// TwinCAT 3 PLC project M3V3_UltraCap
// ProgramVersion: 3.1.4023.0
// libraries:
//   Tc2_Standard, * (Beckhoff Automation GmbH)
//   Tc2_System, * (Beckhoff Automation GmbH)
//   Tc2_Utilities, * (Beckhoff Automation GmbH)
//   Tc3_EventLogger, * (Beckhoff Automation GmbH)
//   Tc3_Module, * (Beckhoff Automation GmbH)
// project tree:
//   DUTs/ E_ChargerType.TcDUT (not stored), E_State.TcDUT (not stored), E_VoltFB.TcDUT (not stored), ST_Alarm_Base.TcDUT (not stored), ST_canRxdata.TcDUT, ST_Cap_Base.TcDUT, ST_Charger_Base.TcDUT, ST_ChargeTime.TcDUT (not stored), ST_MagDriver.TcDUT, ST_Module.TcDUT, ST_PB_Base.TcDUT, ST_Segment_Base.TcDUT, ST_Setpoints_Base.TcDUT, ST_UCDevices.TcDUT, ST_UC_Status.TcDUT, ST_UC_Status_Dummy.TcDUT, ST_UC_Trip_Base.TcDUT, ST_VoltMon_Base.TcDUT (not stored), ST_VoltTran_Base.TcDUT
//   GVLs/ Alarms_DB.TcGVL, ChargeTime_DB.TcGVL, csv_DB.TcGVL (not stored), GVL.TcGVL, plc_plc_comm_DB.TcGVL, HMI_DB.TcGVL, Input.TcGVL, LV.TcGVL, MCP_IO.TcGVL, Output.TcGVL, Permissives_DB.TcGVL, Setpoints.TcGVL, Trips_DB.TcGVL (not stored)
//   / PlcTask.TcTTO (not stored)
//   POUs/ ADC_10V.TcPOU (not stored), ADC_5V.TcPOU (not stored), Alarms.TcPOU, Alarms_FB.TcPOU (not stored), Alias.TcPOU, AnalogConversion.TcPOU, AQ.TcPOU (not stored), CAN_comm.TcPOU, ChargeTime.TcPOU, Heartbeat.TcPOU, HMI.TcPOU, LCA_CAL.TcPOU, MAIN.TcPOU, Norm_x.TcPOU (not stored), Permissives.TcPOU, plc_plc_comm.TcPOU, RW_CSV.TcPOU, Stagger_FB.TcPOU (not stored), Sequence.TcPOU, VoltageMonitor.TcPOU, VoltMonAC_FB.TcPOU (not stored), VoltTranBd.TcPOU
//   POUs/csv/ P_ArgToConvExample.TcPOU, P_StringToConvExample.TcPOU, P_TextModeRead.TcPOU, P_TextModeWrite.TcPOU, P_TextModeWrite_og.TcPOU
// real-time tasks:
//   TASK PlcTask: cycle T#10ms, priority 20, ADS port 350
// I/O:
//   DEVICE Device 3 (EtherCAT), AmsNetId 5.107.220.56.4.1
//     Term 1 (EK1101) [EK1101 EtherCAT Coupler (2A E-Bus, ID switch)]
//       Term 2 (EL3068) [EL3068 8K. Ana. Eingang 0-10V]
//       Term 3 (EL3068) [EL3068 8K. Ana. Eingang 0-10V]
//       Term 4 (EL1008) [EL1008 8Ch. Dig. Input 24V, 3ms]
//       Term 5 (EL1008) [EL1008 8Ch. Dig. Input 24V, 3ms]
//       Term 6 (EL2008) [EL2008 8Ch. Dig. Output 24V, 0.5A]
//       Term 7 (EL2008) [EL2008 8Ch. Dig. Output 24V, 0.5A]
//       Term 8 (EL1008) [EL1008 8Ch. Dig. Input 24V, 3ms]
//       Term 9 (EL2008) [EL2008 8Ch. Dig. Output 24V, 0.5A]
//       Term 10 (EL4008) [EL4008 8Ch. Ana. Output 0-10V, 12bit]
//       Term 21 (EL6751) [EL6751 CANopen Master]
//       Term 22 (EL9011) [EL9011 End Terminal]
//   DEVICE Device 1 (EL6751), AmsNetId 5.107.220.56.2.1
//     Vector__XXX
// variable links:
//   M3V3_UltraCap/M3V3_UltraCap Instance <-> Device 1 (EL6751)/Prepared DBC Signals/Vector__XXX/ElectricalData01
//     PlcTask Inputs/Input.R1_10_CapNumber[1]/Elec_AveVolt <-> Message_Inputs/ELECTRICAL_AVERAGE_VOLTAGE
//     PlcTask Inputs/Input.R1_10_CapNumber[1]/Elec_Balancing <-> Message_Inputs/ELECTRICAL_STATUS_BALANCING
//     PlcTask Inputs/Input.R1_10_CapNumber[1]/Elec_HighestVolt <-> Message_Inputs/ELECTRICAL_HIGHEST_VOLTAGE
//     PlcTask Inputs/Input.R1_10_CapNumber[1]/Elec_Imbalance <-> Message_Inputs/ELECTRICAL_STATUS_IMBALANCE
//     PlcTask Inputs/Input.R1_10_CapNumber[1]/Elec_OverVoltage <-> Message_Inputs/ELECTRICAL_STATUS_OVERVOLTAGE
//     PlcTask Inputs/Input.R1_10_CapNumber[1]/Elec_VoltageSum <-> Message_Inputs/ELECTRICAL_VOLTAGE_SUM
//   M3V3_UltraCap/M3V3_UltraCap Instance <-> Device 1 (EL6751)/Prepared DBC Signals/Vector__XXX/ElectricalData02
//     PlcTask Inputs/Input.R1_10_CapNumber[2]/Elec_AveVolt <-> Message_Inputs/ELECTRICAL_AVERAGE_VOLTAGE
//     PlcTask Inputs/Input.R1_10_CapNumber[2]/Elec_Balancing <-> Message_Inputs/ELECTRICAL_STATUS_BALANCING
//     PlcTask Inputs/Input.R1_10_CapNumber[2]/Elec_HighestVolt <-> Message_Inputs/ELECTRICAL_HIGHEST_VOLTAGE
//     PlcTask Inputs/Input.R1_10_CapNumber[2]/Elec_Imbalance <-> Message_Inputs/ELECTRICAL_STATUS_IMBALANCE
//     PlcTask Inputs/Input.R1_10_CapNumber[2]/Elec_OverVoltage <-> Message_Inputs/ELECTRICAL_STATUS_OVERVOLTAGE
//     PlcTask Inputs/Input.R1_10_CapNumber[2]/Elec_VoltageSum <-> Message_Inputs/ELECTRICAL_VOLTAGE_SUM
//   M3V3_UltraCap/M3V3_UltraCap Instance <-> Device 1 (EL6751)/Prepared DBC Signals/Vector__XXX/ElectricalData03
//     PlcTask Inputs/Input.R1_10_CapNumber[3]/Elec_AveVolt <-> Message_Inputs/ELECTRICAL_AVERAGE_VOLTAGE
//     PlcTask Inputs/Input.R1_10_CapNumber[3]/Elec_Balancing <-> Message_Inputs/ELECTRICAL_STATUS_BALANCING
//     PlcTask Inputs/Input.R1_10_CapNumber[3]/Elec_HighestVolt <-> Message_Inputs/ELECTRICAL_HIGHEST_VOLTAGE
//     PlcTask Inputs/Input.R1_10_CapNumber[3]/Elec_Imbalance <-> Message_Inputs/ELECTRICAL_STATUS_IMBALANCE
//     PlcTask Inputs/Input.R1_10_CapNumber[3]/Elec_OverVoltage <-> Message_Inputs/ELECTRICAL_STATUS_OVERVOLTAGE
//     PlcTask Inputs/Input.R1_10_CapNumber[3]/Elec_VoltageSum <-> Message_Inputs/ELECTRICAL_VOLTAGE_SUM
//   M3V3_UltraCap/M3V3_UltraCap Instance <-> Device 1 (EL6751)/Prepared DBC Signals/Vector__XXX/ElectricalData04
//     PlcTask Inputs/Input.R1_10_CapNumber[4]/Elec_AveVolt <-> Message_Inputs/ELECTRICAL_AVERAGE_VOLTAGE
//     PlcTask Inputs/Input.R1_10_CapNumber[4]/Elec_Balancing <-> Message_Inputs/ELECTRICAL_STATUS_BALANCING
//     PlcTask Inputs/Input.R1_10_CapNumber[4]/Elec_HighestVolt <-> Message_Inputs/ELECTRICAL_HIGHEST_VOLTAGE
//     PlcTask Inputs/Input.R1_10_CapNumber[4]/Elec_Imbalance <-> Message_Inputs/ELECTRICAL_STATUS_IMBALANCE
//     PlcTask Inputs/Input.R1_10_CapNumber[4]/Elec_OverVoltage <-> Message_Inputs/ELECTRICAL_STATUS_OVERVOLTAGE
//     PlcTask Inputs/Input.R1_10_CapNumber[4]/Elec_VoltageSum <-> Message_Inputs/ELECTRICAL_VOLTAGE_SUM
//   M3V3_UltraCap/M3V3_UltraCap Instance <-> Device 1 (EL6751)/Prepared DBC Signals/Vector__XXX/ElectricalData05
//     PlcTask Inputs/Input.R1_10_CapNumber[5]/Elec_AveVolt <-> Message_Inputs/ELECTRICAL_AVERAGE_VOLTAGE
//     PlcTask Inputs/Input.R1_10_CapNumber[5]/Elec_Balancing <-> Message_Inputs/ELECTRICAL_STATUS_BALANCING
//     PlcTask Inputs/Input.R1_10_CapNumber[5]/Elec_HighestVolt <-> Message_Inputs/ELECTRICAL_HIGHEST_VOLTAGE
//     PlcTask Inputs/Input.R1_10_CapNumber[5]/Elec_Imbalance <-> Message_Inputs/ELECTRICAL_STATUS_IMBALANCE
//     PlcTask Inputs/Input.R1_10_CapNumber[5]/Elec_OverVoltage <-> Message_Inputs/ELECTRICAL_STATUS_OVERVOLTAGE
//     PlcTask Inputs/Input.R1_10_CapNumber[5]/Elec_VoltageSum <-> Message_Inputs/ELECTRICAL_VOLTAGE_SUM
//   M3V3_UltraCap/M3V3_UltraCap Instance <-> Device 1 (EL6751)/Prepared DBC Signals/Vector__XXX/ElectricalData06
//     PlcTask Inputs/Input.R1_10_CapNumber[6]/Elec_AveVolt <-> Message_Inputs/ELECTRICAL_AVERAGE_VOLTAGE
//     PlcTask Inputs/Input.R1_10_CapNumber[6]/Elec_Balancing <-> Message_Inputs/ELECTRICAL_STATUS_BALANCING
//     PlcTask Inputs/Input.R1_10_CapNumber[6]/Elec_HighestVolt <-> Message_Inputs/ELECTRICAL_HIGHEST_VOLTAGE
//     PlcTask Inputs/Input.R1_10_CapNumber[6]/Elec_Imbalance <-> Message_Inputs/ELECTRICAL_STATUS_IMBALANCE
//     PlcTask Inputs/Input.R1_10_CapNumber[6]/Elec_OverVoltage <-> Message_Inputs/ELECTRICAL_STATUS_OVERVOLTAGE
//     PlcTask Inputs/Input.R1_10_CapNumber[6]/Elec_VoltageSum <-> Message_Inputs/ELECTRICAL_VOLTAGE_SUM
//   M3V3_UltraCap/M3V3_UltraCap Instance <-> Device 1 (EL6751)/Prepared DBC Signals/Vector__XXX/ElectricalData07
//     PlcTask Inputs/Input.R1_10_CapNumber[7]/Elec_AveVolt <-> Message_Inputs/ELECTRICAL_AVERAGE_VOLTAGE
//     PlcTask Inputs/Input.R1_10_CapNumber[7]/Elec_Balancing <-> Message_Inputs/ELECTRICAL_STATUS_BALANCING
//     PlcTask Inputs/Input.R1_10_CapNumber[7]/Elec_HighestVolt <-> Message_Inputs/ELECTRICAL_HIGHEST_VOLTAGE
//     PlcTask Inputs/Input.R1_10_CapNumber[7]/Elec_Imbalance <-> Message_Inputs/ELECTRICAL_STATUS_IMBALANCE
//     PlcTask Inputs/Input.R1_10_CapNumber[7]/Elec_OverVoltage <-> Message_Inputs/ELECTRICAL_STATUS_OVERVOLTAGE
//     PlcTask Inputs/Input.R1_10_CapNumber[7]/Elec_VoltageSum <-> Message_Inputs/ELECTRICAL_VOLTAGE_SUM
//   M3V3_UltraCap/M3V3_UltraCap Instance <-> Device 1 (EL6751)/Prepared DBC Signals/Vector__XXX/ElectricalData08
//     PlcTask Inputs/Input.R1_10_CapNumber[8]/Elec_AveVolt <-> Message_Inputs/ELECTRICAL_AVERAGE_VOLTAGE
//     PlcTask Inputs/Input.R1_10_CapNumber[8]/Elec_Balancing <-> Message_Inputs/ELECTRICAL_STATUS_BALANCING
//     PlcTask Inputs/Input.R1_10_CapNumber[8]/Elec_HighestVolt <-> Message_Inputs/ELECTRICAL_HIGHEST_VOLTAGE
//     PlcTask Inputs/Input.R1_10_CapNumber[8]/Elec_Imbalance <-> Message_Inputs/ELECTRICAL_STATUS_IMBALANCE
//     PlcTask Inputs/Input.R1_10_CapNumber[8]/Elec_OverVoltage <-> Message_Inputs/ELECTRICAL_STATUS_OVERVOLTAGE
//     PlcTask Inputs/Input.R1_10_CapNumber[8]/Elec_VoltageSum <-> Message_Inputs/ELECTRICAL_VOLTAGE_SUM
//   M3V3_UltraCap/M3V3_UltraCap Instance <-> Device 1 (EL6751)/Prepared DBC Signals/Vector__XXX/ElectricalData09
//     PlcTask Inputs/Input.R1_10_CapNumber[9]/Elec_AveVolt <-> Message_Inputs/ELECTRICAL_AVERAGE_VOLTAGE
//     PlcTask Inputs/Input.R1_10_CapNumber[9]/Elec_Balancing <-> Message_Inputs/ELECTRICAL_STATUS_BALANCING
//     PlcTask Inputs/Input.R1_10_CapNumber[9]/Elec_HighestVolt <-> Message_Inputs/ELECTRICAL_HIGHEST_VOLTAGE
//     PlcTask Inputs/Input.R1_10_CapNumber[9]/Elec_Imbalance <-> Message_Inputs/ELECTRICAL_STATUS_IMBALANCE
//     PlcTask Inputs/Input.R1_10_CapNumber[9]/Elec_OverVoltage <-> Message_Inputs/ELECTRICAL_STATUS_OVERVOLTAGE
//     PlcTask Inputs/Input.R1_10_CapNumber[9]/Elec_VoltageSum <-> Message_Inputs/ELECTRICAL_VOLTAGE_SUM
//   M3V3_UltraCap/M3V3_UltraCap Instance <-> Device 1 (EL6751)/Prepared DBC Signals/Vector__XXX/ElectricalData0A
//     PlcTask Inputs/Input.R1_10_CapNumber[10]/Elec_AveVolt <-> Message_Inputs/ELECTRICAL_AVERAGE_VOLTAGE
//     PlcTask Inputs/Input.R1_10_CapNumber[10]/Elec_Balancing <-> Message_Inputs/ELECTRICAL_STATUS_BALANCING
//     PlcTask Inputs/Input.R1_10_CapNumber[10]/Elec_HighestVolt <-> Message_Inputs/ELECTRICAL_HIGHEST_VOLTAGE
//     PlcTask Inputs/Input.R1_10_CapNumber[10]/Elec_Imbalance <-> Message_Inputs/ELECTRICAL_STATUS_IMBALANCE
//     PlcTask Inputs/Input.R1_10_CapNumber[10]/Elec_OverVoltage <-> Message_Inputs/ELECTRICAL_STATUS_OVERVOLTAGE
//     PlcTask Inputs/Input.R1_10_CapNumber[10]/Elec_VoltageSum <-> Message_Inputs/ELECTRICAL_VOLTAGE_SUM
//   M3V3_UltraCap/M3V3_UltraCap Instance <-> Device 1 (EL6751)/Prepared DBC Signals/Vector__XXX/ElectricalData0B
//     PlcTask Inputs/Input.R1_10_CapNumber[11]/Elec_AveVolt <-> Message_Inputs/ELECTRICAL_AVERAGE_VOLTAGE
//     PlcTask Inputs/Input.R1_10_CapNumber[11]/Elec_Balancing <-> Message_Inputs/ELECTRICAL_STATUS_BALANCING
//     PlcTask Inputs/Input.R1_10_CapNumber[11]/Elec_HighestVolt <-> Message_Inputs/ELECTRICAL_HIGHEST_VOLTAGE
//     PlcTask Inputs/Input.R1_10_CapNumber[11]/Elec_Imbalance <-> Message_Inputs/ELECTRICAL_STATUS_IMBALANCE
//     PlcTask Inputs/Input.R1_10_CapNumber[11]/Elec_OverVoltage <-> Message_Inputs/ELECTRICAL_STATUS_OVERVOLTAGE
//     PlcTask Inputs/Input.R1_10_CapNumber[11]/Elec_VoltageSum <-> Message_Inputs/ELECTRICAL_VOLTAGE_SUM
//   M3V3_UltraCap/M3V3_UltraCap Instance <-> Device 1 (EL6751)/Prepared DBC Signals/Vector__XXX/ElectricalData0C
//     PlcTask Inputs/Input.R1_10_CapNumber[12]/Elec_AveVolt <-> Message_Inputs/ELECTRICAL_AVERAGE_VOLTAGE
//     PlcTask Inputs/Input.R1_10_CapNumber[12]/Elec_Balancing <-> Message_Inputs/ELECTRICAL_STATUS_BALANCING
//     PlcTask Inputs/Input.R1_10_CapNumber[12]/Elec_HighestVolt <-> Message_Inputs/ELECTRICAL_HIGHEST_VOLTAGE
//     PlcTask Inputs/Input.R1_10_CapNumber[12]/Elec_Imbalance <-> Message_Inputs/ELECTRICAL_STATUS_IMBALANCE
//     PlcTask Inputs/Input.R1_10_CapNumber[12]/Elec_OverVoltage <-> Message_Inputs/ELECTRICAL_STATUS_OVERVOLTAGE
//     PlcTask Inputs/Input.R1_10_CapNumber[12]/Elec_VoltageSum <-> Message_Inputs/ELECTRICAL_VOLTAGE_SUM
//   M3V3_UltraCap/M3V3_UltraCap Instance <-> Device 1 (EL6751)/Prepared DBC Signals/Vector__XXX/ElectricalData7F
//     PlcTask Inputs/Input.R1_10_UC_7F_status/Elec_AveVolt <-> Message_Inputs/ELECTRICAL_AVERAGE_VOLTAGE
//     PlcTask Inputs/Input.R1_10_UC_7F_status/Elec_Balancing <-> Message_Inputs/ELECTRICAL_STATUS_BALANCING
//     PlcTask Inputs/Input.R1_10_UC_7F_status/Elec_HighestVolt <-> Message_Inputs/ELECTRICAL_HIGHEST_VOLTAGE
//     PlcTask Inputs/Input.R1_10_UC_7F_status/Elec_Imbalance <-> Message_Inputs/ELECTRICAL_STATUS_IMBALANCE
//     PlcTask Inputs/Input.R1_10_UC_7F_status/Elec_OverVoltage <-> Message_Inputs/ELECTRICAL_STATUS_OVERVOLTAGE
//     PlcTask Inputs/Input.R1_10_UC_7F_status/Elec_VoltageSum <-> Message_Inputs/ELECTRICAL_VOLTAGE_SUM
//   M3V3_UltraCap/M3V3_UltraCap Instance <-> Device 1 (EL6751)/Prepared DBC Signals/Vector__XXX/ThermalData01
//     PlcTask Inputs/Input.R1_10_CapNumber[1]/Therm_HighestCell <-> Message_Inputs/THERMAL_HIGHEST_CELL
//     PlcTask Inputs/Input.R1_10_CapNumber[1]/Therm_LowestCell <-> Message_Inputs/THERMAL_LOWEST_CELL
//   M3V3_UltraCap/M3V3_UltraCap Instance <-> Device 1 (EL6751)/Prepared DBC Signals/Vector__XXX/ThermalData02
//     PlcTask Inputs/Input.R1_10_CapNumber[2]/Therm_HighestCell <-> Message_Inputs/THERMAL_HIGHEST_CELL
//     PlcTask Inputs/Input.R1_10_CapNumber[2]/Therm_LowestCell <-> Message_Inputs/THERMAL_LOWEST_CELL
//   M3V3_UltraCap/M3V3_UltraCap Instance <-> Device 1 (EL6751)/Prepared DBC Signals/Vector__XXX/ThermalData03
//     PlcTask Inputs/Input.R1_10_CapNumber[3]/Therm_HighestCell <-> Message_Inputs/THERMAL_HIGHEST_CELL
//     PlcTask Inputs/Input.R1_10_CapNumber[3]/Therm_LowestCell <-> Message_Inputs/THERMAL_LOWEST_CELL
//   M3V3_UltraCap/M3V3_UltraCap Instance <-> Device 1 (EL6751)/Prepared DBC Signals/Vector__XXX/ThermalData04
//     PlcTask Inputs/Input.R1_10_CapNumber[4]/Therm_HighestCell <-> Message_Inputs/THERMAL_HIGHEST_CELL
//     PlcTask Inputs/Input.R1_10_CapNumber[4]/Therm_LowestCell <-> Message_Inputs/THERMAL_LOWEST_CELL
//   M3V3_UltraCap/M3V3_UltraCap Instance <-> Device 1 (EL6751)/Prepared DBC Signals/Vector__XXX/ThermalData05
//     PlcTask Inputs/Input.R1_10_CapNumber[5]/Therm_HighestCell <-> Message_Inputs/THERMAL_HIGHEST_CELL
//     PlcTask Inputs/Input.R1_10_CapNumber[5]/Therm_LowestCell <-> Message_Inputs/THERMAL_LOWEST_CELL
//   M3V3_UltraCap/M3V3_UltraCap Instance <-> Device 1 (EL6751)/Prepared DBC Signals/Vector__XXX/ThermalData06
//     PlcTask Inputs/Input.R1_10_CapNumber[6]/Therm_HighestCell <-> Message_Inputs/THERMAL_HIGHEST_CELL
//     PlcTask Inputs/Input.R1_10_CapNumber[6]/Therm_LowestCell <-> Message_Inputs/THERMAL_LOWEST_CELL
//   M3V3_UltraCap/M3V3_UltraCap Instance <-> Device 1 (EL6751)/Prepared DBC Signals/Vector__XXX/ThermalData07
//     PlcTask Inputs/Input.R1_10_CapNumber[7]/Therm_HighestCell <-> Message_Inputs/THERMAL_HIGHEST_CELL
//     PlcTask Inputs/Input.R1_10_CapNumber[7]/Therm_LowestCell <-> Message_Inputs/THERMAL_LOWEST_CELL
//   M3V3_UltraCap/M3V3_UltraCap Instance <-> Device 1 (EL6751)/Prepared DBC Signals/Vector__XXX/ThermalData08
//     PlcTask Inputs/Input.R1_10_CapNumber[8]/Therm_HighestCell <-> Message_Inputs/THERMAL_HIGHEST_CELL
//     PlcTask Inputs/Input.R1_10_CapNumber[8]/Therm_LowestCell <-> Message_Inputs/THERMAL_LOWEST_CELL
//   M3V3_UltraCap/M3V3_UltraCap Instance <-> Device 1 (EL6751)/Prepared DBC Signals/Vector__XXX/ThermalData09
//     PlcTask Inputs/Input.R1_10_CapNumber[9]/Therm_HighestCell <-> Message_Inputs/THERMAL_HIGHEST_CELL
//     PlcTask Inputs/Input.R1_10_CapNumber[9]/Therm_LowestCell <-> Message_Inputs/THERMAL_LOWEST_CELL
//   M3V3_UltraCap/M3V3_UltraCap Instance <-> Device 1 (EL6751)/Prepared DBC Signals/Vector__XXX/ThermalData0A
//     PlcTask Inputs/Input.R1_10_CapNumber[10]/Therm_HighestCell <-> Message_Inputs/THERMAL_HIGHEST_CELL
//     PlcTask Inputs/Input.R1_10_CapNumber[10]/Therm_LowestCell <-> Message_Inputs/THERMAL_LOWEST_CELL
//   M3V3_UltraCap/M3V3_UltraCap Instance <-> Device 1 (EL6751)/Prepared DBC Signals/Vector__XXX/ThermalData0B
//     PlcTask Inputs/Input.R1_10_CapNumber[11]/Therm_HighestCell <-> Message_Inputs/THERMAL_HIGHEST_CELL
//     PlcTask Inputs/Input.R1_10_CapNumber[11]/Therm_LowestCell <-> Message_Inputs/THERMAL_LOWEST_CELL
//   M3V3_UltraCap/M3V3_UltraCap Instance <-> Device 1 (EL6751)/Prepared DBC Signals/Vector__XXX/ThermalData0C
//     PlcTask Inputs/Input.R1_10_CapNumber[12]/Therm_HighestCell <-> Message_Inputs/THERMAL_HIGHEST_CELL
//     PlcTask Inputs/Input.R1_10_CapNumber[12]/Therm_LowestCell <-> Message_Inputs/THERMAL_LOWEST_CELL
//   M3V3_UltraCap/M3V3_UltraCap Instance <-> Device 1 (EL6751)/Prepared DBC Signals/Vector__XXX/ThermalData7F
//     PlcTask Inputs/Input.R1_10_UC_7F_status/Therm_HighestCell <-> Message_Inputs/THERMAL_HIGHEST_CELL
//     PlcTask Inputs/Input.R1_10_UC_7F_status/Therm_LowestCell <-> Message_Inputs/THERMAL_LOWEST_CELL
//   M3V3_UltraCap/M3V3_UltraCap Instance <-> Device 3 (EtherCAT)/Term 1 (EK1101)/Term 10 (EL4008)
//     PlcTask Outputs/Output.R1_09_00 <-> AO Outputs Channel 1/Analog output
//     PlcTask Outputs/Output.R1_09_01 <-> AO Outputs Channel 2/Analog output
//     PlcTask Outputs/Output.R1_09_02 <-> AO Outputs Channel 3/Analog output
//     PlcTask Outputs/Output.R1_09_03 <-> AO Outputs Channel 4/Analog output
//     PlcTask Outputs/Output.R1_09_04 <-> AO Outputs Channel 5/Analog output
//     PlcTask Outputs/Output.R1_09_05 <-> AO Outputs Channel 6/Analog output
//     PlcTask Outputs/Output.R1_09_06 <-> AO Outputs Channel 7/Analog output
//     PlcTask Outputs/Output.R1_09_07 <-> AO Outputs Channel 8/Analog output
//   M3V3_UltraCap/M3V3_UltraCap Instance <-> Device 3 (EtherCAT)/Term 1 (EK1101)/Term 2 (EL3068)
//     PlcTask Inputs/Input.R1_01_00 <-> AI Standard Channel 1/Value
//     PlcTask Inputs/Input.R1_01_01 <-> AI Standard Channel 2/Value
//     PlcTask Inputs/Input.R1_01_02 <-> AI Standard Channel 3/Value
//     PlcTask Inputs/Input.R1_01_03 <-> AI Standard Channel 4/Value
//     PlcTask Inputs/Input.R1_01_04 <-> AI Standard Channel 5/Value
//     PlcTask Inputs/Input.R1_01_05 <-> AI Standard Channel 6/Value
//     PlcTask Inputs/Input.R1_01_06 <-> AI Standard Channel 7/Value
//     PlcTask Inputs/Input.R1_01_07 <-> AI Standard Channel 8/Value
//   M3V3_UltraCap/M3V3_UltraCap Instance <-> Device 3 (EtherCAT)/Term 1 (EK1101)/Term 3 (EL3068)
//     PlcTask Inputs/Input.R1_02_00 <-> AI Standard Channel 1/Value
//     PlcTask Inputs/Input.R1_02_01 <-> AI Standard Channel 2/Value
//     PlcTask Inputs/Input.R1_02_02 <-> AI Standard Channel 3/Value
//     PlcTask Inputs/Input.R1_02_03 <-> AI Standard Channel 4/Value
//     PlcTask Inputs/Input.R1_02_04 <-> AI Standard Channel 5/Value
//     PlcTask Inputs/Input.R1_02_05 <-> AI Standard Channel 6/Value
//     PlcTask Inputs/Input.R1_02_06 <-> AI Standard Channel 7/Value
//     PlcTask Inputs/Input.R1_02_07 <-> AI Standard Channel 8/Value
//   M3V3_UltraCap/M3V3_UltraCap Instance <-> Device 3 (EtherCAT)/Term 1 (EK1101)/Term 4 (EL1008)
//     PlcTask Inputs/Input.R1_03_00 <-> Channel 1/Input
//     PlcTask Inputs/Input.R1_03_01 <-> Channel 2/Input
//     PlcTask Inputs/Input.R1_03_02 <-> Channel 3/Input
//     PlcTask Inputs/Input.R1_03_03 <-> Channel 4/Input
//     PlcTask Inputs/Input.R1_03_04 <-> Channel 5/Input
//     PlcTask Inputs/Input.R1_03_05 <-> Channel 6/Input
//     PlcTask Inputs/Input.R1_03_06 <-> Channel 7/Input
//     PlcTask Inputs/Input.R1_03_07 <-> Channel 8/Input
//   M3V3_UltraCap/M3V3_UltraCap Instance <-> Device 3 (EtherCAT)/Term 1 (EK1101)/Term 5 (EL1008)
//     PlcTask Inputs/Input.R1_04_00 <-> Channel 1/Input
//     PlcTask Inputs/Input.R1_04_01 <-> Channel 2/Input
//     PlcTask Inputs/Input.R1_04_02 <-> Channel 3/Input
//     PlcTask Inputs/Input.R1_04_03 <-> Channel 4/Input
//     PlcTask Inputs/Input.R1_04_04 <-> Channel 5/Input
//     PlcTask Inputs/Input.R1_04_05 <-> Channel 6/Input
//     PlcTask Inputs/Input.R1_04_06 <-> Channel 7/Input
//     PlcTask Inputs/Input.R1_04_07 <-> Channel 8/Input
//   M3V3_UltraCap/M3V3_UltraCap Instance <-> Device 3 (EtherCAT)/Term 1 (EK1101)/Term 6 (EL2008)
//     PlcTask Outputs/Output.R1_05_00 <-> Channel 1/Output
//     PlcTask Outputs/Output.R1_05_01 <-> Channel 2/Output
//     PlcTask Outputs/Output.R1_05_02 <-> Channel 3/Output
//     PlcTask Outputs/Output.R1_05_03 <-> Channel 4/Output
//     PlcTask Outputs/Output.R1_05_04 <-> Channel 5/Output
//     PlcTask Outputs/Output.R1_05_05 <-> Channel 6/Output
//     PlcTask Outputs/Output.R1_05_06 <-> Channel 7/Output
//     PlcTask Outputs/Output.R1_05_07 <-> Channel 8/Output
//   M3V3_UltraCap/M3V3_UltraCap Instance <-> Device 3 (EtherCAT)/Term 1 (EK1101)/Term 7 (EL2008)
//     PlcTask Outputs/Output.R1_06_00 <-> Channel 1/Output
//     PlcTask Outputs/Output.R1_06_01 <-> Channel 2/Output
//     PlcTask Outputs/Output.R1_06_02 <-> Channel 3/Output
//     PlcTask Outputs/Output.R1_06_03 <-> Channel 4/Output
//     PlcTask Outputs/Output.R1_06_04 <-> Channel 5/Output
//     PlcTask Outputs/Output.R1_06_05 <-> Channel 6/Output
//     PlcTask Outputs/Output.R1_06_06 <-> Channel 7/Output
//     PlcTask Outputs/Output.R1_06_07 <-> Channel 8/Output
//   M3V3_UltraCap/M3V3_UltraCap Instance <-> Device 3 (EtherCAT)/Term 1 (EK1101)/Term 8 (EL1008)
//     PlcTask Inputs/Input.R1_07_00 <-> Channel 1/Input
//     PlcTask Inputs/Input.R1_07_01 <-> Channel 2/Input
//     PlcTask Inputs/Input.R1_07_02 <-> Channel 3/Input
//     PlcTask Inputs/Input.R1_07_03 <-> Channel 4/Input
//     PlcTask Inputs/Input.R1_07_04 <-> Channel 5/Input
//     PlcTask Inputs/Input.R1_07_05 <-> Channel 6/Input
//     PlcTask Inputs/Input.R1_07_06 <-> Channel 7/Input
//     PlcTask Inputs/Input.R1_07_07 <-> Channel 8/Input
//   M3V3_UltraCap/M3V3_UltraCap Instance <-> Device 3 (EtherCAT)/Term 1 (EK1101)/Term 9 (EL2008)
//     PlcTask Outputs/Output.R1_08_00 <-> Channel 1/Output
//     PlcTask Outputs/Output.R1_08_01 <-> Channel 2/Output
//     PlcTask Outputs/Output.R1_08_02 <-> Channel 3/Output
//     PlcTask Outputs/Output.R1_08_03 <-> Channel 4/Output
//     PlcTask Outputs/Output.R1_08_04 <-> Channel 5/Output
//     PlcTask Outputs/Output.R1_08_05 <-> Channel 6/Output
//     PlcTask Outputs/Output.R1_08_06 <-> Channel 7/Output
//     PlcTask Outputs/Output.R1_08_07 <-> Channel 8/Output

// ---- DUTs/ST_canRxdata.TcDUT
TYPE ST_canRxdata :
STRUCT
	cobID			: STRING;
	deviceID		: ARRAY [1..12] OF STRING; // will make it 1..10 later
	byteData		: ARRAY [0..7] OF USINT;
	byteData_hexstr	: ARRAY [0..7] OF STRING;
END_STRUCT
END_TYPE

// ---- DUTs/ST_Cap_Base.TcDUT
TYPE ST_Cap_Base :
STRUCT
	
	CapWarning			: BOOL;  //comes from UltraCaps CANBUS message
	CapAlarm			: BOOL;
	CapVoltage			: REAL;   //Comes from UlgraCaps CANBUS message
	CapCellTemp			: REAL;
	
	//UltraCap_CAN_ID : STRING;
	Elec_Balancing		: USINT;
	Elec_Imbalance		: USINT;
	Elec_VoltageSum		: LREAL;
	Elec_HighestVolt	: LREAL;
	Elec_AveVolt		: LREAL;
	Elec_OverVoltage	: USINT;
	
	Therm_LowTemp		: USINT;
	Therm_HighTemp		: USINT;
	Therm_HighestCell	: LREAL;
	Therm_LowestCell	: LREAL;
	
	//UltraCap			: ST_UC_Status;  //assuming 10 uc in one coil
	UltraCap_Dummy		: ST_UC_Status_Dummy; //buffer temp for uc 7f
	UC_Dummy_ID_hexstr	: STRING;
	
	CanTx_config_ID 	: UDINT;
	CanTx_config_length : UINT;
	CanTx_config_request: ARRAY[0..7] OF BYTE;
END_STRUCT
END_TYPE

// ---- DUTs/ST_Charger_Base.TcDUT
TYPE ST_Charger_Base :
STRUCT
	//DI
	//inhibited 		: BOOL;
	OverTemp		: BOOL;
	DCOK			: BOOL;
	ACOK			: BOOL;
	
	//DQ
	inhibit			: BOOL;
	
	//AI
	(*voltageFeedback_raw 	: INT;
	voltageFeedback_norm 	: REAL;
	voltageFeedback			: REAL;
	
	currentFeedback_raw 	: INT;
	currentFeedback_norm	: REAL;
	currentFeedback			: REAL;
	*)
	//AQ
	voltageSP_norm	: REAL;
	voltageSP		: REAL; // **V
	voltageSP_raw	: INT; // setpoint output to field device.
	//internal 
	ChargeTime		: ST_ChargeTime;
END_STRUCT
END_TYPE

// ---- DUTs/ST_MagDriver.TcDUT
TYPE ST_MagDriver :
STRUCT
	SCR_ready_to_fire 		: BOOL := FALSE;
	ChargeRelayClose		: BOOL := FALSE;
	DumpRelayOpen			: BOOL := FALSE;
	
	CloseChargeRly			: BOOL := FALSE;
	OpenDumpRly				: BOOL := FALSE;
	
	DumpResistorTemp_raw	: INT;
	DumpResistorTemp_norm	: REAL;
	DumpResistorTemp		: REAL;
	
	ShotCurrentFeedback_raw	: INT;
	ShotCurrentFeedback_norm: REAL;
	ShotCurrentFeedback		: REAL;
	
	//Charger 				: ST_Charger_Base; //MCP IO alreayd hs it

	Cap						: ARRAY[1..2] OF ST_Cap_Base;

END_STRUCT
END_TYPE

// ---- DUTs/ST_Module.TcDUT
TYPE ST_Module :
STRUCT
	//DumpRly_close	: BOOL;
	
	VoltageFeedback : ARRAY[1..2] OF REAL;
	VoltageFeedback_norm : ARRAY[1..2] OF REAL;
	VoltageFeedback_raw : ARRAY[1..2] OF DINT;
	//VTB : ARRAY[1..2] OF ST_VoltTran_Base;  uncomment this for troubleshooting the bits in VoltageMonitor POU
END_STRUCT
END_TYPE

// ---- DUTs/ST_PB_Base.TcDUT
TYPE ST_PB_Base :
STRUCT
	FirePBPressed : BOOL := FALSE;
	spare1	: BOOL := FALSE;
	spare2	: BOOL := FALSE;
	spare3	: BOOL := FALSE;
	spare4	: BOOL := FALSE;
	spare5	: BOOL := FALSE;
	spare6	: BOOL := FALSE;
	spare7	: BOOL := FALSE;
	spare8	: BOOL := FALSE;
	spare9	: BOOL := FALSE;
	spare10	: BOOL := FALSE;
	spare11	: BOOL := FALSE;
	spare12	: BOOL := FALSE;
	spare13	: BOOL := FALSE;
	spare14	: BOOL := FALSE;
	spare15	: BOOL := FALSE;
END_STRUCT
END_TYPE

// ---- DUTs/ST_Segment_Base.TcDUT
TYPE ST_Segment_Base :
STRUCT
	Module : ARRAY [1..9] OF ST_Module;	
	
	CloseChargeRly	: BOOL;
	ChargeRly_close : BOOL;

	OpenModule1To3DumpRly : BOOL; //Open Module1To3DumpRly
	OpenModule4To6DumpRly : BOOL;
	OpenModule7To9DumpRly : BOOL;
	
	Module1To3DumpRly_close	: BOOL;
	Module4To6DumpRly_close	: BOOL;
	Module7To9DumpRly_close	: BOOL;
	//ShortContactClose	: BOOL;

END_STRUCT
END_TYPE

// ---- DUTs/ST_Setpoints_Base.TcDUT
TYPE ST_Setpoints_Base :
STRUCT
	RequiredChargedV : REAL := 105;
	TotalCapacitance : REAL := 10; //uF - LOCAL ONLY, NOT FROM MAIN PLC - LoadCapacitance
	ChargeTime		 : REAL := 360; //6min charge time
	//PSratedV		 : REAL := 50;
	//wLCA			 : BOOL := TRUE;
	//NumOfCharger	 : INT := 2;
	//eChargerType		: E_ChargerType;
END_STRUCT
END_TYPE

// ---- DUTs/ST_UCDevices.TcDUT
TYPE ST_UCDevices :
STRUCT
	//Status : ST_UC_Status; - obsolete
	Elec_Balancing		: USINT;
	Elec_Imbalance		: USINT;
	Elec_VoltageSum		: LREAL;
	Elec_HighestVolt	: LREAL;
	Elec_AveVolt		: LREAL;
	Elec_OverVoltage	: USINT;
	
	Therm_LowTemp		: USINT;
	Therm_HighTemp		: USINT;
	Therm_HighestCell	: LREAL;
	Therm_LowestCell	: LREAL;
END_STRUCT
END_TYPE

// ---- DUTs/ST_UC_Status.TcDUT
TYPE ST_UC_Status :
STRUCT
	Elec_Balancing		: USINT;
	Elec_Imbalance		: USINT;
	Elec_VoltageSum		: LREAL;
	Elec_HighestVolt	: LREAL;
	Elec_AveVolt		: LREAL;
	Elec_OverVoltage	: USINT;
	
	Therm_LowTemp		: USINT;
	Therm_HighTemp		: USINT;
	Therm_HighestCell	: LREAL;
	Therm_LowestCell	: LREAL;
	
END_STRUCT
END_TYPE

// ---- DUTs/ST_UC_Status_Dummy.TcDUT
TYPE ST_UC_Status_Dummy EXTENDS ST_UC_Status :
STRUCT
	R1_10_UC_Rx_cobID : UDINT;
	R1_10_UC_Rx_data : ARRAY [0..7] OF BYTE;
END_STRUCT
END_TYPE

// ---- DUTs/ST_UC_Trip_Base.TcDUT
TYPE ST_UC_Trip_Base :
STRUCT
	UC_Cell_OverV_StatusError	: BOOL; //0x11
	UC_Cell_OverV_warning		: BOOL; //0x01 
	UC_Cell_OverV_alarm			: BOOL; //0x10
	
	UC_tempHigh_StatusError		: BOOL; //0x11
	UC_tempHigh_warning			: BOOL; //0x01
	UC_tempHigh_alarm			: BOOL; //0x10
END_STRUCT
END_TYPE

// ---- DUTs/ST_VoltTran_Base.TcDUT
TYPE ST_VoltTran_Base :
STRUCT
	BateryLow 			: BOOL := 0;
	VoltageReading_raw	: INT; //custom board
	CapRaw				: UINT;
	DataNull			: BOOL := 0;
	LossVoltTransBoard	: BOOL := 0;
END_STRUCT
END_TYPE

// ---- GVLs/Alarms_DB.TcGVL
{attribute 'qualified_only'}
VAR_GLOBAL
	MCP	: ST_Alarm_Base;
	Segment1 : ST_Alarm_Base;
	
	AlarmWord1  : ST_Alarm_Base;
	AlarmWord2  : ST_Alarm_Base;
	AlarmWord3  : ST_Alarm_Base;

END_VAR

// ---- GVLs/ChargeTime_DB.TcGVL
{attribute 'qualified_only'}
VAR_GLOBAL RETAIN
	ChargerDelay_TON : ARRAY[1..6] OF TON;
	ChargerDelay_PT  : ARRAY[1..6] OF TIME;
	ChargerDelay_ET  : ARRAY[1..6] OF TIME;	
	
	//SustChargeTime_TON : ARRAY[1..3] OF TON;
	//SustChargeTime_PT  : ARRAY[1..3] OF TIME;
	//SustChargeTime_ET  : ARRAY[1..3] OF TIME;	
	
	//FormChargeTime_TON : ARRAY[1..2] OF TON;
	//FormChargeTime_PT  : ARRAY[1..2] OF TIME;
	//FormChargeTime_ET  : ARRAY[1..2] OF TIME;
	
	PreFormChargeTime_TON : TON;
	PreFormChargeTime_PT : TIME;
	PreFormChargeTime_ET : TIME;
	
	LongestChargeTime_TON : TON;
	LongestChargeTime_PT : TIME;
	LongestChargeTime_ET : TIME;

	ChargeTimeStartDelay	: ARRAY[1..6] OF INT;
	ChargingTimeElapse		: ARRAY[1..6] OF INT;	
	ChargingTimeElapse_TON	: ARRAY[1..6] OF TON;

END_VAR

// ---- GVLs/GVL.TcGVL
{attribute 'qualified_only'}
VAR_GLOBAL
END_VAR

VAR_GLOBAL CONSTANT
	MAX_CSV_ROWS 			: UDINT := 500;
	MAX_CSV_COLUMNS 		: UDINT := 6; // 0 - 6, so 7
	MAX_CSV_FIELD_LENGTH	: UDINT := 150;
END_VAR

// ---- GVLs/plc_plc_comm_DB.TcGVL
{attribute 'qualified_only'}
VAR_GLOBAL
	ReadStateFromPLC	AT %MB0 : E_State; // 1 = p1 comp pp charge complete, 2 = p1 comp pp dumping
	WriteStatetoPLC		AT %MB2	: E_State;
	
	ChargeTime 		AT %MB4 : REAL; //send charge time m1 pp
	
	Button 			AT %MB8	: ST_PB_Base;	// %MB ; 4020, %MX; 4021
END_VAR

// ---- GVLs/HMI_DB.TcGVL
{attribute 'qualified_only'}
VAR_GLOBAL PERSISTENT
	HPT5		: ARRAY [1..6] OF ST_Setpoints_Base; //or RETAIN
	
	ChargerHVOFF_rlyDelayPT		: TIME := T#25MS;
	ChargerHVOFF_rlyDelayPT_INT	: INT := 25;
	
	HVONdelayPT					: TIME := T#250MS;
	HVONdelayPT_INT				: INT := 250;
	
	RunOutTMR_PT				: TIME := T#10S;
	RunOutTMR_PT_INT			: DINT := 10;
	RunOutTMR_elapse			: DINT;
	
	ChargingRunOutTMR_elapse	: INT;
	DumpResTempThres			: UINT := 125;
	
	CAN_Comm_MagDriverNum		: INT := 1;
	CAN_Comm_UC_Num				: INT := 1;
		
END_VAR

VAR_GLOBAL
	ArmTheCagePB				: BOOL := 0;
	UnArmTheCagePB				: BOOL := 0;
	ChargePB					: BOOL := 0;
	DumpPB						: BOOL := 0;
	AbortPB						: BOOL := 0;
	FirePB						: BOOL := 0;
	ClearFaultPB				: BOOL := 0;
	AllDumpRelaysOpenBP			: BOOL := 0;
	AllChargeRelayCloseBP		: BOOL := 0;
	SystemSafeBP				: BOOL := 0;
	ForceToChargCompletePB		: BOOL := 0;
	
	HMI_ManualModeSelected		: BOOL := 0;  // 1 = manual mode selected
	CloseChargeRlySW			: BOOL := 0;
	OpenDumpRlySW				: BOOL := 0;
	TurnChrgHVonSW				: BOOL := 0;
	TurnChrgInhibitOffSW		: BOOL := 0;
	TurnOnShotTrigSW			: BOOL := 0;
	TurnOnChargeAlarm			: BOOL := 0;
	
	LastTimeShotLog				: BOOL := 0;
	CSV_loggingBusy				: BOOL := 0;
	CSV_loggingError			: BOOL := 0;
	CSV_loggingDone				: BOOL := 0;
	FillingBuffer				: BOOL := 0;
	AllCapsDischargedBP			: BOOL := FALSE;
	
END_VAR

// ---- GVLs/Input.TcGVL
{attribute 'qualified_only'}
VAR_GLOBAL
//***MCP************************************************************************

//EL3068 - AI1
	R1_01_00 		AT %I*: INT;
	R1_01_00_Status AT %I*: WORD;
	R1_01_01 		AT %I*: INT;
	R1_01_01_Status AT %I*: WORD;
	R1_01_02 		AT %I*: INT;
	R1_01_02_Status AT %I*: WORD;
	R1_01_03 		AT %I*: INT;
	R1_01_03_Status AT %I*: WORD;
	R1_01_04 		AT %I*: INT;
	R1_01_04_Status AT %I*: WORD;
	R1_01_05 		AT %I*: INT;
	R1_01_05_Status AT %I*: WORD;
	R1_01_06 		AT %I*: INT;
	R1_01_06_Status AT %I*: WORD;
	R1_01_07 		AT %I*: INT;
	R1_01_07_Status AT %I*: WORD;

	//EL3068 - AI2
	R1_02_00 		AT %I*: INT;
	R1_02_00_Status AT %I*: WORD;
	R1_02_01 		AT %I*: INT;
	R1_02_01_Status AT %I*: WORD;
	R1_02_02 		AT %I*: INT;
	R1_02_02_Status AT %I*: WORD;
	R1_02_03 		AT %I*: INT;
	R1_02_03_Status AT %I*: WORD;
	R1_02_04 		AT %I*: INT;
	R1_02_04_Status AT %I*: WORD;
	R1_02_05 		AT %I*: INT;
	R1_02_05_Status AT %I*: WORD;
	R1_02_06 		AT %I*: INT;
	R1_02_06_Status AT %I*: WORD;
	R1_02_07 		AT %I*: INT;
	R1_02_07_Status AT %I*: WORD;
	
	//EL1008 - DI1
	R1_03_00 AT	%I*: BOOL; //Master stop PB not pressed - black pb on mcp
	R1_03_01 AT	%I*: BOOL; //case Estop circuit okay (Rly1 (120vac)
	R1_03_02 AT %I*: BOOL; //MCP PSU1 DC OK
	R1_03_03 AT %I*: BOOL; //
	R1_03_04 AT %I*: BOOL; //
	R1_03_05 AT %I*: BOOL; //spare
	R1_03_06 AT %I*: BOOL; //spare
	R1_03_07 AT %I*: BOOL; //spare
	
	//EL1008 - DI2
	R1_04_00 AT	%I*: BOOL;  
	R1_04_01 AT	%I*: BOOL;
	R1_04_02 AT %I*: BOOL; 
	R1_04_03 AT %I*: BOOL; 
	R1_04_04 AT %I*: BOOL; 
	R1_04_05 AT %I*: BOOL; 
	R1_04_06 AT %I*: BOOL; 
	R1_04_07 AT %I*: BOOL; 
	
	//EL1008 - DI3
	R1_07_00 AT	%I*: BOOL;  
	R1_07_01 AT	%I*: BOOL;
	R1_07_02 AT %I*: BOOL; 
	R1_07_03 AT %I*: BOOL; 
	R1_07_04 AT %I*: BOOL; 
	R1_07_05 AT %I*: BOOL; 
	R1_07_06 AT %I*: BOOL; 
	R1_07_07 AT %I*: BOOL;
	
	//add CANbus
	
	//Ethercat Device Voltage - subject to change because the VM board is still under development
	(*B170357_CapRaw AT %I* : ARRAY[0..24] OF UINT;
	B170357_BatLevel AT %I* : BOOL;
	B170357_Heartbeat AT %I* : BOOL;*)

	R1_10_CapNumber AT %I* : ARRAY [1..12] OF  ST_UC_Status; //only used with DBC file.
	R1_10_UC_7F_status AT %I* : ST_UC_Status_Dummy;
	R1_10_UC_status AT %I* : ARRAY [1..12] OF ST_UC_Status_Dummy;

	
END_VAR

// ---- GVLs/LV.TcGVL
{attribute 'qualified_only'}
VAR_GLOBAL
	TxWord1	: WORD; // received PB from LV
	TxWord2 : WORD;
	TxWord3 : WORD;
	
	RxWord1 : WORD; 
	RxWord2 : WORD;
	RxWord3 : WORD;

	
	TxInt : ARRAY [1..5] OF INT;
	TxDint : ARRAY [1..3] OF DINT;
	TxREAL : ARRAY [1..12] OF REAL;

	RxInt : ARRAY [1..2] OF INT;
	RxDint : ARRAY [1..3] OF DINT;
	RxREAL : ARRAY [1..18] OF REAL;
	
	Charger : ARRAY[1..7] OF ST_Charger_Base;
	
	HPT5Load	: ARRAY [1..7] OF ST_Setpoints_Base; 
	ReadState		: E_State;
	WriteState		: E_State;
	
	database		: ARRAY[0..GVL.MAX_CSV_ROWS, 0..GVL.MAX_CSV_COLUMNS ] OF STRING(GVL.MAX_CSV_FIELD_LENGTH) :=[ (* Source PLC database *)
	'0_0', '0_1', '0_2', '0_3', '0_4', '0_5', '0_6',
	'1_0', '1_1', '1_2', '1_3', '1_4', '1_5', '1_6',
	'2_0', '2_1', '2_2', '2_3', '2_4', '2_5', '2_6',
	'3_0', '3_1', '3_2', '3_3', '3_4', '3_5', '3_6',
	'4_0', '4_1', '4_2', '4_3', '4_4', '4_5', '4_6',
	'5_0', '5_1', '5_2', '5_3', '5_4', '5_5', '5_6'];
	(*ChargerHVOFF_rlyDelayPT		: TIME := T#25MS;
	ChargerHVOFF_rlyDelayPT_INT	: INT := 25;
	
	HVONdelayPT					: TIME := T#250MS;
	HVONdelayPT_INT				: INT := 250;
	
	RunOutTMR_PT				: TIME := T#10S;
	RunOutTMR_PT_INT			: DINT := 10;
	RunOutTMR_elapse			: DINT;
	
	ChargingRunOutTMR_elapse	: INT;
	
	ChargePB					: BOOL := 0;
	DumpPB						: BOOL := 0;
	AbortPB						: BOOL := 0;
	FirePB						: BOOL := 0;
	ClearFaultPB				: BOOL := 0;
	AllDumpRelaysOpenBP			: BOOL := 0;
	AllChargeRelayCloseBP		: BOOL := 0;
	SystemSafeBP				: BOOL := 0;
	
	HMI_ManualModeSelected		: BOOL := 0;  // 1 = manual mode selected
	CloseChargeRlySW			: BOOL := 0;
	OpenDumpRlySW				: BOOL := 0;*)
END_VAR

// ---- GVLs/MCP_IO.TcGVL
{attribute 'qualified_only'}
VAR_GLOBAL
	MasterStopPB_NotPressed		: BOOL := FALSE;
	CageEstopCircuitOK			: BOOL := FALSE;
	//RemoteModeSelected			: BOOL;
	PSU1_DCOK					: BOOL;
	MagDriver					: ARRAY[1..6] OF ST_MagDriver;
	TriggerSCRs					: BOOL := FALSE;
	TriggerScope				: BOOL := FALSE;
	TurnONSystemChargedLED		: BOOL := FALSE;
	
	//Cap							: ARRAY[1..12] OF ST_Cap_Base;	
	

	//MachineGNDrlyOpen			: BOOL;
	//CloseAllChargeRlyCommand	: BOOL; only for slim
	//OpenAllDumpRelayCommand		: BOOL; only for slim
	//Charger 					: ARRAY [1..8] OF ST_Charger_Base;
	//GLS3_Load					: ST_ChargeTime;
	//GLS1_hvON					: BOOL;
	//GLS2_hvON					: BOOL;
	//GLS3_hvON					: BOOL;
	//LiftMachineGND				: BOOL;
	//AllChargeRelaysClose		: BOOL; only for slim
	//AllDumpRelaysOpen			: BOOL; only for slim
	//GLS1_voltageSP				: DINT;
	//GLS1_voltageSP_norm			: REAL;
	//GLS1_voltageSP_raw			: INT;
	
	//GLS2_voltageSP				: DINT;
	//GLS2_voltageSP_norm			: REAL;
	//GLS2_voltageSP_raw			: INT;
	
	//GLS3_voltageSP				: DINT;
	//GLS3_voltageSP_norm			: REAL;
	//GLS3_voltageSP_raw			: INT;

END_VAR

VAR_GLOBAL PERSISTENT
	Charger 					: ARRAY [1..6] OF ST_Charger_Base;
END_VAR

// ---- GVLs/Output.TcGVL
{attribute 'qualified_only'}
VAR_GLOBAL
//***MCP 
	//EL2008 - DQ1
	R1_05_00 AT %Q*: BOOL;
	R1_05_01 AT %Q*: BOOL;
	R1_05_02 AT %Q*: BOOL;
	R1_05_03 AT %Q*: BOOL;
	R1_05_04 AT %Q*: BOOL;
	R1_05_05 AT %Q*: BOOL;
	R1_05_06 AT %Q*: BOOL;
	R1_05_07 AT %Q*: BOOL;
	
	//EL2008 - DQ2
	R1_06_00 AT %Q*: BOOL;
	R1_06_01 AT %Q*: BOOL;
	R1_06_02 AT %Q*: BOOL;
	R1_06_03 AT %Q*: BOOL;
	R1_06_04 AT %Q*: BOOL;
	R1_06_05 AT %Q*: BOOL;
	R1_06_06 AT %Q*: BOOL;
	R1_06_07 AT %Q*: BOOL;
	
	//EL2008 - DQ3
	R1_08_00 AT %Q*: BOOL;
	R1_08_01 AT %Q*: BOOL;
	R1_08_02 AT %Q*: BOOL;
	R1_08_03 AT %Q*: BOOL;
	R1_08_04 AT %Q*: BOOL;
	R1_08_05 AT %Q*: BOOL;
	R1_08_06 AT %Q*: BOOL;
	R1_08_07 AT %Q*: BOOL;
	
	//EL4008 - AQ1
	R1_09_00 AT %Q*: INT;	//Charger 1 - Voltage Setpoint
	R1_09_01 AT %Q*: INT;	//Charger 2 - Voltage Setpoint
	R1_09_02 AT %Q*: INT;	//Charger 3 - Voltage Setpoint
	R1_09_03 AT %Q*: INT;	//Charger 4 - Voltage Setpoint
	R1_09_04 AT %Q*: INT;	//Charger 5 - Voltage Setpoint	
	R1_09_05 AT %Q*: INT;	//Charger 6 - Voltage Setpoint	
	R1_09_06 AT %Q*: INT;	//spare
	R1_09_07 AT %Q*: INT;	//spare
	
	R1_10_7F_CANrequest AT %Q*: EXTCANQUEUE; //this one is for 7F
	R1_10_ARR_CANrequest AT %Q*: ARRAY [1..12] OF EXTCANQUEUE ;	
	
END_VAR

// ---- GVLs/Permissives_DB.TcGVL
{attribute 'qualified_only'}
VAR_GLOBAL
	//SafetyOK				: BOOL;
	AllChargeRelayClosed 	: BOOL := FALSE;
	AllDumpRelayOpen		: BOOL := FALSE;
	//AllDumpRelayClose		: BOOL := 0;
	ReadyToCharge			: BOOL := FALSE;
	//AllChargerEOC			: BOOL := FALSE;
	
	ChargerVBelowThres		: BOOL := FALSE;
	ChargerVThres			: REAL := 10;
	AllChargerDCOK			: BOOL := FALSE;
	AllChargerACOK			: BOOL := FALSE;
	AllChargerInhibitON		: BOOL := 0;

	AllCapsDischarged		: BOOL := FALSE;
	CapVoltageThres			: REAL := 40;
	
	AllChargerTempOK		: BOOL := FALSE;
	TempThres				: REAL := 50;
	AllDumpResTempOK		: BOOL := FALSE;

	SystemIsSafe			: BOOL := FALSE;
	AllSCRreadyToFire		: BOOL := FALSE;
END_VAR

// ---- GVLs/Setpoints.TcGVL
{attribute 'qualified_only'}
VAR_GLOBAL
	HPT5 : ARRAY [1..7] OF ST_Setpoints_Base;

	
END_VAR

// ---- POUs/ChargeTime.TcPOU
PROGRAM ChargeTime
VAR

	//lca_charge_cal	 : ARRAY [1..6] OF LCA_CAL;
	i				 : INT := 1; // 1-6 instances
	j				 : INT := 1; //1 - 6 ch
	m				 : INT := 1;
	n				 : INT := 6;
	a				 : INT := 1; 
	
	Q				 : REAL := 1; // Charge
	Current			 : REAL := 0.1; //100mA
	
	longestChargeTime: REAL;
	
END_VAR

//mapping hmi input to setpoints
FOR j := 1 TO n BY 1 DO	
	Setpoints.HPT5[j].TotalCapacitance	:= HMI_DB.HPT5[j].TotalCapacitance;
	//Setpoints.TDKLoad[j].PSratedV 			:= HMI_DB.TDKLoad[j].PSratedV;
	Setpoints.HPT5[j].RequiredChargedV	:= HMI_DB.HPT5[j].RequiredChargedV;  
	//Setpoints.TDKLoad[j].wLCA				:= HMI_DB.TDKLoad[j].wLCA;
	//Setpoints.TDKLoad[j].NumOfCharger		:= HMI_DB.TDKLoad[j].NumOfCharger;	
	
	//charge time delay and elapse for HMI
	ChargeTime_DB.ChargeTimeStartDelay[j] := TIME_TO_INT((ChargeTime_DB.ChargerDelay_PT[j] - ChargeTime_DB.ChargerDelay_ET[j])/1000);
	ChargeTime_DB.ChargingTimeElapse[j] := TIME_TO_INT((ChargeTime_DB.ChargingTimeElapse_TON[j].PT - ChargeTime_DB.ChargingTimeElapse_TON[j].ET)/1000);
END_FOR

//ChargeTime_DB.PreFormChargeTimeStartDelay := TIME_TO_INT((ChargeTime_DB.PreFormChargeTime_PT - ChargeTime_DB.PreFormChargeTime_ET)/1000);
//ChargeTime_DB.PreFormChargingTimeElapse := TIME_TO_INT((ChargeTime_DB.PreFormChargingTimeElapse_TON.PT - ChargeTime_DB.PreFormChargingTimeElapse_TON.ET)/1000);

(*
//GLS 3
Setpoints.GLSLoad.TotalCapacitance	:= HMI_DB.GLSLoad.TotalCapacitance;
Setpoints.GLSLoad.PSratedV 			:= HMI_DB.GLSLoad.PSratedV;
//Setpoints.PreFormBank.RequiredChargedV	:= Recipe.PreFormBank.RequiredChargedV; //only thing that comes from the main plc recipe
//Setpoints.GLSLoad.wLCA				:= HMI_DB.GLSLoad.wLCA;
Setpoints.GLSLoad.NumOfCharger		:= HMI_DB.GLSLoad.NumOfCharger;	
*)


//veto
//this should not happen
FOR m := 1 TO n BY 1 DO
	IF Setpoints.HPT5[m].RequiredChargedV <= -1 THEN
		Setpoints.HPT5[m].RequiredChargedV := 0;
	END_IF	
END_FOR

FOR i := 1 TO n BY 1 DO
	//set limites of charger voltage input from HMI input
	IF (Setpoints.HPT5[i].RequiredChargedV) >= AnalogConversion.MaxVolt THEN
		Setpoints.HPT5[i].RequiredChargedV := AnalogConversion.MaxVolt; //limit at 105v
		HMI_DB.HPT5[i].RequiredChargedV := AnalogConversion.MaxVolt;
	ELSIF Setpoints.HPT5[i].RequiredChargedV <= 0 THEN
		Setpoints.HPT5[i].RequiredChargedV := 0;
		HMI_DB.HPT5[i].RequiredChargedV := 0;
	END_IF	
END_FOR;

//chg time
FOR i := 1 TO n BY 1 DO
	//manually enter charge time*********************
	MCP_IO.Charger[i].ChargeTime.timeToChargeLoad := HMI_DB.HPT5[i].ChargeTime;
	
	IF Setpoints.HPT5[i].RequiredChargedV = 0 THEN
		MCP_IO.Charger[i].ChargeTime.timeToChargeLoad := 0;
		MCP_IO.Charger[i].ChargeTime.Power := 0;
	END_IF
END_FOR

(*
//gls - gls3 is preform cap charger
Q := 1000* Setpoints.GLSLoad.RequiredChargedV * (Setpoints.GLSLoad.TotalCapacitance / 1000000);
MCP_IO.GLS3_Load.timeToChargeLoad := Q / Current;
MCP_IO.GLS3_Load.Power := 1000*Setpoints.GLSLoad.RequiredChargedV * Current;
*)

//find the longest charge time.  //need more work
longestChargeTime := MAX( MCP_IO.Charger[1].ChargeTime.timeToChargeLoad,
							MCP_IO.Charger[2].ChargeTime.timeToChargeLoad,
							MCP_IO.Charger[3].ChargeTime.timeToChargeLoad,
							MCP_IO.Charger[4].ChargeTime.timeToChargeLoad,
							MCP_IO.Charger[5].ChargeTime.timeToChargeLoad,
							MCP_IO.Charger[6].ChargeTime.timeToChargeLoad);

ChargeTime_DB.LongestChargeTime_PT := REAL_TO_TIME (1000*longestChargeTime);

plc_plc_comm_DB.ChargeTime := longestChargeTime; //send charge time to m1 pp

//FOR a := 1 TO 8 BY 1 DO
FOR a := 1 TO n BY 1 DO
	IF (longestChargeTime - MCP_IO.Charger[a].ChargeTime.timeToChargeLoad) >= 0 THEN
		ChargeTime_DB.ChargerDelay_PT[a] := REAL_TO_TIME (1000*(longestChargeTime - MCP_IO.Charger[a].ChargeTime.timeToChargeLoad));
		ELSE 
			ChargeTime_DB.ChargerDelay_PT[a] := REAL_TO_TIME (1000*(MCP_IO.Charger[a].ChargeTime.timeToChargeLoad - longestChargeTime));
	END_IF;		
		
	//IF (longestChargeTime - MCP_IO.Charger[a+3].ChargeTime.timeToChargeLoad) >= 0 THEN
	//	ChargeTime_DB.SustChargeTime_PT[a] := REAL_TO_TIME (1000*(longestChargeTime - MCP_IO.Charger[a+3].ChargeTime.timeToChargeLoad));	
	//END_IF;	
	
END_FOR;


(*IF (longestChargeTime - MCP_IO.Charger[7].ChargeTime.timeToChargeLoad) >= 0 THEN
	ChargeTime_DB.FormChargeTime_PT[1] := REAL_TO_TIME (1000*(longestChargeTime - MCP_IO.Charger[7].ChargeTime.timeToChargeLoad));	
END_IF;	
IF (longestChargeTime - MCP_IO.Charger[8].ChargeTime.timeToChargeLoad) >= 0 THEN
	ChargeTime_DB.FormChargeTime_PT[2] := REAL_TO_TIME (1000*(longestChargeTime - MCP_IO.Charger[8].ChargeTime.timeToChargeLoad));	
END_IF;	

IF (longestChargeTime - MCP_IO.GLS3_Load.timeToChargeLoad) >= 0 THEN
		ChargeTime_DB.PreFormChargeTime_PT := REAL_TO_TIME (1000*(longestChargeTime - MCP_IO.GLS3_Load.timeToChargeLoad));
		ELSE
			ChargeTime_DB.PreFormChargeTime_PT := REAL_TO_TIME (1000*(MCP_IO.GLS3_Load.timeToChargeLoad -longestChargeTime));
END_IF;
*)



IF i > n THEN 
	i := 1;
END_IF

IF j > n THEN
	j := 1;
END_IF

IF m > n THEN
	m := 1;
END_IF


IF a > n THEN
	a := 1;
END_IF;

END_PROGRAM

// ---- POUs/AnalogConversion.TcPOU
PROGRAM AnalogConversion
VAR
	i					: INT := 1; //charger 1-6
	j					: INT := 1;  // section 1 - 4 
	k					: INT := 1;  // cap 1-10
	m					: INT := 1; //form cap 1-12
	n					: INT := 6;
	MaxTemp				: INT := 380;
	MinTemp				: INT := -70;
	
	MaxCurrent			: INT := 1000;
	MinCurrent			: INT := 0;
	
	MaxVolt				: INT := 105;
	//VoltMonAC1			: ARRAY[1..18] OF VoltMonAC_FB;
	//VoltMonAC2			: ARRAY[1..18] OF VoltMonAC_FB;
END_VAR

//MCP Charger 
//Analog Input
FOR i := 1 TO n BY 1 DO 
	//MCP_IO.Charger[i].voltageSP := (HMI_DB.TDKLoad[i].RequiredChargedV *1000);
	MCP_IO.Charger[i].voltageSP := (Setpoints.HPT5[i].RequiredChargedV);
END_FOR

//AI
FOR i := 1 TO n BY 1 DO
	//Temp
	MCP_IO.MagDriver[i].DumpResistorTemp_norm := Norm_x (raw_input := INT_TO_REAL (MCP_IO.MagDriver[i].DumpResistorTemp_raw),
														x_max := 32767,
														x_min := 6553); // temp sensor is 4-20mA
											
	MCP_IO.MagDriver[i].DumpResistorTemp := (MaxTemp - MinTemp) * ADC_10V( normal_input := MCP_IO.MagDriver[i].DumpResistorTemp_norm,
																			x_max := 10,
																			x_min := 2); // temp sensor is 2-10v
	//current																									
	MCP_IO.MagDriver[i].ShotCurrentFeedback_norm := Norm_x (raw_input := INT_TO_REAL (MCP_IO.MagDriver[i].ShotCurrentFeedback_raw),
														x_max := 32767,
														x_min := 0);
	
	MCP_IO.MagDriver[1].ShotCurrentFeedback := (MaxCurrent - MinCurrent) * ADC_10V( normal_input := MCP_IO.MagDriver[i].ShotCurrentFeedback_norm,
																							x_max := 10,
																							x_min := 0);

END_FOR;

//Analog Output
//voltageSP = Required Charge Voltage******************
//limit for charing the cap
//FOR i := 1 TO 8 BY 1 DO
FOR i := 1 TO n BY 1 DO	
	
	//set limits of charger voltage input 
	IF MCP_IO.Charger[i].voltageSP >= (MaxVolt) THEN
		MCP_IO.Charger[i].voltageSP := MaxVolt; //limit at 105V
	ELSIF MCP_IO.Charger[i].voltageSP <= 0 THEN
		MCP_IO.Charger[i].voltageSP := 0; //limit at 0V
	END_IF; 
		
	//prepare output signal for 50kV chargers.
	MCP_IO.Charger[i].voltageSP_norm := Norm_x (raw_input :=(MCP_IO.Charger[i].voltageSP), 
												x_max := MaxVolt,
												x_min := 0);	
												
	MCP_IO.Charger[i].voltageSP_raw := AQ (norm_input := MCP_IO.Charger[i].voltageSP_norm, 
												x_max := 20,
												x_min := 0);
																								
	//limite for output sigal (<= 10V)  this should not happen
	IF MCP_IO.Charger[i].voltageSP_raw >= (32767/2) THEN //32767/2
		MCP_IO.Charger[i].voltageSP_raw := (32767/2); 										
	END_IF;
	
END_FOR;

//no need for cap voltage feedback - the ultacap already scale those internally

//Cap voltage feedback
(*
//can also add a range of x samples for self calibrating **note: normalized range needs to be calibrated for each board
VoltMonitor_DB.VoltageReading_norm[0] := Norm_x (raw_input := INT_TO_REAL (VoltMonitor_DB.VoltageReading_raw[0]),
													x_max := 904, //10bit value - 1110001000 = 904deci
													x_min := 100); //100deci is the zero of range -1.61 to 12.01
LCP1_IO.Segment[1].Module[1].VoltageFeedback[1] := (12010 - 0) * ADC_10V(normal_input := VoltMonitor_DB.VoltageReading_norm[0],
																		x_max := 12.01,
																		x_min := 0); //use zero, it will cal for the -ve	

*)

(* // changed to a FB for norm and ADC
LCP1_IO.Segment[1].Module[1].VoltageFeedback_norm[1] := Norm_x (raw_input := INT_TO_REAL (LCP1_IO.Segment[1].Module[1].VoltageFeedback_raw[1]),
													x_max := 904, //10bit value - 1110001000 = 904deci
													x_min := 100); //100deci is the zero of range -1.61 to 12.01
LCP1_IO.Segment[1].Module[1].VoltageFeedback[1] := (12010 - 0) * ADC_10V(normal_input := LCP1_IO.Segment[1].Module[1].VoltageFeedback_norm[1],
																		x_max := 12.01,
																		x_min := 0); //use zero, it will cal for the -ve
*)

(*
// using FB instead.
VoltMonAC1[1](raw_input := DINT_TO_REAL(LCP1_IO.Segment[1].Module[1].VoltageFeedback_raw[1]),
				norm_x_max := 904, //individually calibrated, otherwise can do a for loop
				norm_x_min := 100, 
				RangUpp := 12.01, 
				RangLow := 0, 
				ADC_max := 12010, 
				ADC_min := 0, 
				voltage_reading => LCP1_IO.Segment[1].Module[1].VoltageFeedback[1]);
*)

					
//reset counter
//IF i > 8 THEN
IF i > n THEN
	i := 1;
END_IF;

IF j > 3 THEN 
	j := 1;
END_IF

IF k > 10 THEN 
	k := 1;
END_IF

IF m > 12 THEN 
	m := 1;
END_IF

END_PROGRAM

// ---- POUs/Alarms.TcPOU
PROGRAM Alarms
VAR
	bWarning : BOOL;
	bConfirm : BOOL;
	alarms : ARRAY[0..32] OF Alarms_FB;
	
END_VAR

// Alarm Word 1 - MCP Alarms
//MCP Alarms - need to modify this for pfc

Alarms_DB.MCP.AlarmWord.0 := Trips_DB.AnyEstopPressed;
Alarms_DB.MCP.AlarmWord.1 := Trips_DB.CageDoorNotClose;
Alarms_DB.MCP.AlarmWord.2 := Trips_DB.ShortingSystemUnknown;
//Alarms_DB.MCP.AlarmWord.3 := 
//Alarms_DB.MCP.AlarmWord.4 := MCP_IO.Charger[1].SummaryFaulted;
//Alarms_DB.MCP.AlarmWord.5 := MCP_IO.Charger[2].SummaryFaulted;
//Alarms_DB.MCP.AlarmWord.6 := MCP_IO.Charger[3].SummaryFaulted;
//Alarms_DB.MCP.AlarmWord.7 := MCP_IO.Charger[4].SummaryFaulted;
//Alarms_DB.MCP.AlarmWord.8 := MCP_IO.Charger[5].SummaryFaulted;
//Alarms_DB.MCP.AlarmWord.9 := MCP_IO.Charger[6].SummaryFaulted;
Alarms_DB.MCP.AlarmWord.10 := HMI_DB.ForceToChargCompletePB;
//Alarms_DB.MCP.AlarmWord.11 := VoltMonitor_DB.LossVoltMonitorBoard;
Alarms_DB.MCP.AlarmWord.12 := Trips_DB.ChargedTimerRunout;
Alarms_DB.MCP.AlarmWord.13 := Trips_DB.ChargingTimerRunout;
Alarms_DB.MCP.AlarmWord.14 := HMI_DB.LastTimeShotLog;
//Alarms_DB.MCP.AlarmWord.15 := HMI.ForceCharCompSatisfied;

//Alarm Word 1 msg
//IE: alarms[299](evtEntry:= Tc_Events.AlarmWord11.b4, bEvt:= gvl.test, bConfirm:= bConfirm);
alarms[0](evtEntry:= Tc_Events.AlarmWord1.b0, bEvt:= Alarms_DB.MCP.AlarmWord.0, bConfirm:= bConfirm);
alarms[1](evtEntry:= Tc_Events.AlarmWord1.b1, bEvt:= Alarms_DB.MCP.AlarmWord.1, bConfirm:= bConfirm);
alarms[2](evtEntry:= Tc_Events.AlarmWord1.b2, bEvt:= Alarms_DB.MCP.AlarmWord.2, bConfirm:= bConfirm);
alarms[3](evtEntry:= Tc_Events.AlarmWord1.b3, bEvt:= Alarms_DB.MCP.AlarmWord.3, bConfirm:= bConfirm);
alarms[4](evtEntry:= Tc_Events.AlarmWord1.b4, bEvt:= Alarms_DB.MCP.AlarmWord.4, bConfirm:= bConfirm);
alarms[5](evtEntry:= Tc_Events.AlarmWord1.b5, bEvt:= Alarms_DB.MCP.AlarmWord.5, bConfirm:= bConfirm);
alarms[6](evtEntry:= Tc_Events.AlarmWord1.b6, bEvt:= Alarms_DB.MCP.AlarmWord.6, bConfirm:= bConfirm);
alarms[7](evtEntry:= Tc_Events.AlarmWord1.b7, bEvt:= Alarms_DB.MCP.AlarmWord.7, bConfirm:= bConfirm);
alarms[8](evtEntry:= Tc_Events.AlarmWord1.b8, bEvt:= Alarms_DB.MCP.AlarmWord.8, bConfirm:= bConfirm);
alarms[9](evtEntry:= Tc_Events.AlarmWord1.b9, bEvt:= Alarms_DB.MCP.AlarmWord.9, bConfirm:= bConfirm);
alarms[0](evtEntry:= Tc_Events.AlarmWord1.b10, bEvt:= Alarms_DB.MCP.AlarmWord.10, bConfirm:= bConfirm);
alarms[11](evtEntry:= Tc_Events.AlarmWord1.b11, bEvt:= Alarms_DB.MCP.AlarmWord.11, bConfirm:= bConfirm);
alarms[12](evtEntry:= Tc_Events.AlarmWord1.b12, bEvt:= Alarms_DB.MCP.AlarmWord.12, bConfirm:= bConfirm);
alarms[13](evtEntry:= Tc_Events.AlarmWord1.b13, bEvt:= Alarms_DB.MCP.AlarmWord.13, bConfirm:= bConfirm);
alarms[14](evtEntry:= Tc_Events.AlarmWord1.b14, bEvt:= Alarms_DB.MCP.AlarmWord.14, bConfirm:= bConfirm);
alarms[15](evtEntry:= Tc_Events.AlarmWord1.b15, bEvt:= Alarms_DB.MCP.AlarmWord.15, bConfirm:= bConfirm);

// Alarm Word 2 - Section 1 Alarms
(*Alarms_DB.Section1.AlarmWord.0 := Trips_DB.Section[1].SystemTripped;
Alarms_DB.Section1.AlarmWord.1 := Trips_DB.Section[1].LossPneumaticPressure;
Alarms_DB.Section1.AlarmWord.2 := Trips_DB.Section[1].Peak.ChargeRelay1_Failed;
Alarms_DB.Section1.AlarmWord.3 := Trips_DB.Section[1].Peak.ChargeRelay2_Failed;
Alarms_DB.Section1.AlarmWord.4 := Trips_DB.Section[1].Peak.DumpRelay1_Failed;
Alarms_DB.Section1.AlarmWord.5 := Trips_DB.Section[1].Peak.DumpRelay2_Failed;
Alarms_DB.Section1.AlarmWord.6 := Trips_DB.Section[1].Sust.ChargeRelay1_Failed;
Alarms_DB.Section1.AlarmWord.7 := Trips_DB.Section[1].Sust.ChargeRelay2_Failed;
Alarms_DB.Section1.AlarmWord.8 := Trips_DB.Section[1].Sust.DumpRelay1_Failed;
Alarms_DB.Section1.AlarmWord.9 := Trips_DB.Section[1].Sust.DumpRelay2_Failed;
Alarms_DB.Section1.AlarmWord.10 := Trips_DB.Section[1].LossDCPower;


// Alarm Word 2 - Msg
alarms[16](evtEntry:= Tc_Events.AlarmWord2.b0, bEvt:= Alarms_DB.Section1.AlarmWord.0, bConfirm:= bConfirm);
alarms[17](evtEntry:= Tc_Events.AlarmWord2.b1, bEvt:= Alarms_DB.Section1.AlarmWord.1, bConfirm:= bConfirm);
alarms[18](evtEntry:= Tc_Events.AlarmWord2.b2, bEvt:= Alarms_DB.Section1.AlarmWord.2, bConfirm:= bConfirm);
alarms[19](evtEntry:= Tc_Events.AlarmWord2.b3, bEvt:= Alarms_DB.Section1.AlarmWord.3, bConfirm:= bConfirm);
alarms[20](evtEntry:= Tc_Events.AlarmWord2.b4, bEvt:= Alarms_DB.Section1.AlarmWord.4, bConfirm:= bConfirm);
alarms[21](evtEntry:= Tc_Events.AlarmWord2.b5, bEvt:= Alarms_DB.Section1.AlarmWord.5, bConfirm:= bConfirm);
alarms[22](evtEntry:= Tc_Events.AlarmWord2.b6, bEvt:= Alarms_DB.Section1.AlarmWord.6, bConfirm:= bConfirm);
alarms[23](evtEntry:= Tc_Events.AlarmWord2.b7, bEvt:= Alarms_DB.Section1.AlarmWord.7, bConfirm:= bConfirm);
alarms[24](evtEntry:= Tc_Events.AlarmWord2.b8, bEvt:= Alarms_DB.Section1.AlarmWord.8, bConfirm:= bConfirm);
alarms[25](evtEntry:= Tc_Events.AlarmWord2.b9, bEvt:= Alarms_DB.Section1.AlarmWord.9, bConfirm:= bConfirm);
alarms[26](evtEntry:= Tc_Events.AlarmWord2.b10, bEvt:= Alarms_DB.Section1.AlarmWord.10, bConfirm:= bConfirm);
//alarms[27] - spare
//alarms[28] - spare
//alarms[29] - spare
//alarms[30] - spare
//alarms[31] - spare
*)

//Clear Alarm Word
IF bConfirm THEN
	Alarms_DB.MCP.AlarmWord := 0;
	Alarms_DB.Segment1.AlarmWord := 0;
	
	(*Alarms_DB.Coil3.AlarmWord := 0;
	Alarms_DB.Coil4.AlarmWord := 0;
	Alarms_DB.Coil5.AlarmWord := 0;
	Alarms_DB.Coil6.AlarmWord := 0;
	Alarms_DB.Coil7.AlarmWord := 0;
	Alarms_DB.Coil8.AlarmWord := 0;
	Alarms_DB.Coil9.AlarmWord := 0;
	Alarms_DB.Coil10.AlarmWord := 0;
	Alarms_DB.AlarmWord_11.AlarmWord := 0;
	Alarms_DB.AlarmWord_22.AlarmWord := 0;
	Alarms_DB.AlarmWord_23.AlarmWord := 0;
	Alarms_DB.AlarmWord_24.AlarmWord := 0;
	Alarms_DB.AlarmWord_25.AlarmWord := 0;
	Alarms_DB.AlarmWord_26.AlarmWord := 0;
	Alarms_DB.AlarmWord_27.AlarmWord := 0;
	*)
END_IF;

END_PROGRAM

// ---- POUs/Alias.TcPOU
PROGRAM Alias
VAR
	i : INT := 1; //mag driver index
	n : INT := 6; //mag driver num
	j : INT := 1; //1-2
	m : INT := 2; //# of ultra cap per driver rack
	k : INT := 1; //ultra cap number 

	
	p : INT := 12; //# of ultra caps = 12
	
END_VAR

//R1 : MCP**  
	//INPUT
	//AI - EL3068
	MCP_IO.MagDriver[1].ShotCurrentFeedback_raw	:= Input.R1_01_00; //
	MCP_IO.MagDriver[2].ShotCurrentFeedback_raw	:= Input.R1_01_01; //
	MCP_IO.MagDriver[3].ShotCurrentFeedback_raw	:= Input.R1_01_02; // 
	MCP_IO.MagDriver[4].ShotCurrentFeedback_raw	:= Input.R1_01_03; //
	MCP_IO.MagDriver[5].ShotCurrentFeedback_raw	:= Input.R1_01_04; // 
	MCP_IO.MagDriver[6].ShotCurrentFeedback_raw	:= Input.R1_01_05; //  
	//Spare										:= Input.R1_01_06; //  
	//Spare										:= Input.R1_01_07; //
	
	//DI
	MCP_IO.MagDriver[1].DumpResistorTemp_raw	:= Input.R1_02_00; //
	MCP_IO.MagDriver[2].DumpResistorTemp_raw	:= Input.R1_02_01; // 
	MCP_IO.MagDriver[3].DumpResistorTemp_raw	:= Input.R1_02_02; // 
	MCP_IO.MagDriver[4].DumpResistorTemp_raw	:= Input.R1_02_03; // 
	MCP_IO.MagDriver[5].DumpResistorTemp_raw	:= Input.R1_02_04; // 
	MCP_IO.MagDriver[6].DumpResistorTemp_raw	:= Input.R1_02_05; // 
	
	MCP_IO.MagDriver[1].SCR_ready_to_fire		:= Input.R1_03_00; // 
	MCP_IO.MagDriver[2].SCR_ready_to_fire		:= Input.R1_03_01; // 
	MCP_IO.MagDriver[3].SCR_ready_to_fire		:= Input.R1_03_02; // 
	MCP_IO.MagDriver[4].SCR_ready_to_fire		:= Input.R1_03_03; // 
	MCP_IO.MagDriver[5].SCR_ready_to_fire		:= Input.R1_03_04; // 
	MCP_IO.MagDriver[6].SCR_ready_to_fire		:= Input.R1_03_05; // 
	
	MCP_IO.MagDriver[1].ChargeRelayClose		:= Input.R1_04_00; //
	MCP_IO.MagDriver[2].ChargeRelayClose		:= Input.R1_04_01; //
	MCP_IO.MagDriver[3].ChargeRelayClose		:= Input.R1_04_02; //
	MCP_IO.MagDriver[4].ChargeRelayClose		:= Input.R1_04_03; //
	MCP_IO.MagDriver[5].ChargeRelayClose		:= Input.R1_04_04; //
	MCP_IO.MagDriver[6].ChargeRelayClose		:= Input.R1_04_05; //
	
	//DQ
	Output.R1_05_00	:= MCP_IO.MagDriver[1].CloseChargeRly;
	Output.R1_05_01	:= MCP_IO.MagDriver[2].CloseChargeRly;
	Output.R1_05_02	:= MCP_IO.MagDriver[3].CloseChargeRly;
	Output.R1_05_03	:= MCP_IO.MagDriver[4].CloseChargeRly;
	Output.R1_05_04	:= MCP_IO.MagDriver[5].CloseChargeRly;
	Output.R1_05_05	:= MCP_IO.MagDriver[6].CloseChargeRly;
	//Output.R1_05_06	:= 
	//Output.R1_05_07	:= 
	
	//DQ
	Output.R1_06_00	:= MCP_IO.MagDriver[1].OpenDumpRly;
	Output.R1_06_01	:= MCP_IO.MagDriver[2].OpenDumpRly;
	Output.R1_06_02	:= MCP_IO.MagDriver[3].OpenDumpRly;
	Output.R1_06_03	:= MCP_IO.MagDriver[4].OpenDumpRly;
	Output.R1_06_04 := MCP_IO.MagDriver[5].OpenDumpRly;
	Output.R1_06_05 := MCP_IO.MagDriver[6].OpenDumpRly;
	
	MCP_IO.MagDriver[1].DumpRelayOpen		:= NOT Input.R1_07_00; //
	MCP_IO.MagDriver[2].DumpRelayOpen		:= NOT Input.R1_07_01; //
	MCP_IO.MagDriver[3].DumpRelayOpen		:= NOT Input.R1_07_02; //
	MCP_IO.MagDriver[4].DumpRelayOpen		:= NOT Input.R1_07_03; //
	MCP_IO.MagDriver[5].DumpRelayOpen		:= NOT Input.R1_07_04; //
	MCP_IO.MagDriver[6].DumpRelayOpen		:= NOT Input.R1_07_05; //
	(*shaft ramp add below*)
	
	//DQ
	Output.R1_08_00	:= NOT MCP_IO.Charger[1].inhibit;
	Output.R1_08_01	:= NOT MCP_IO.Charger[2].inhibit;
	Output.R1_08_02	:= NOT MCP_IO.Charger[3].inhibit;
	Output.R1_08_03	:= NOT MCP_IO.Charger[4].inhibit;
	Output.R1_08_04	:= NOT MCP_IO.Charger[5].inhibit;
	Output.R1_08_05	:= NOT MCP_IO.Charger[6].inhibit;
	Output.R1_08_06 := MCP_IO.TriggerSCRs;
	Output.R1_08_07	:= MCP_IO.TurnONSystemChargedLED;
		
	//EL4008 AQ
	Output.R1_09_00	:= MCP_IO.Charger[1].voltageSP_raw;
	Output.R1_09_01	:= MCP_IO.Charger[2].voltageSP_raw;
	Output.R1_09_02	:= MCP_IO.Charger[3].voltageSP_raw;
	Output.R1_09_03	:= MCP_IO.Charger[4].voltageSP_raw;	
	Output.R1_09_04	:= MCP_IO.Charger[5].voltageSP_raw;
	Output.R1_09_05	:= MCP_IO.Charger[6].voltageSP_raw;
	
	//CANBUS 
	//Output.R1_10_CANrequest := CAN_comm. ---delete, this is 7F
	Output.R1_10_7F_CANrequest.cobId := CAN_comm.CanTx_7F_config_ID;
	Output.R1_10_7F_CANrequest.data[0] := CAN_comm.CanTx_7F_config_request[0];
	Output.R1_10_7F_CANrequest.data[1] := CAN_comm.CanTx_7F_config_request[1];
	Output.R1_10_7F_CANrequest.data[2] := CAN_comm.CanTx_7F_config_request[2];
	Output.R1_10_7F_CANrequest.data[3] := CAN_comm.CanTx_7F_config_request[3];
	Output.R1_10_7F_CANrequest.data[4] := CAN_comm.CanTx_7F_config_request[4];
	Output.R1_10_7F_CANrequest.data[5] := CAN_comm.CanTx_7F_config_request[5];
	Output.R1_10_7F_CANrequest.data[6] := CAN_comm.CanTx_7F_config_request[6];
	Output.R1_10_7F_CANrequest.data[7] := CAN_comm.CanTx_7F_config_request[7];
	
		//will eventually need to make a loop for this - code below
	Output.R1_10_ARR_CANrequest[1].cobId := MCP_IO.MagDriver[1].Cap[1].CanTx_config_ID;
	Output.R1_10_ARR_CANrequest[1].data[0] := MCP_IO.MagDriver[1].Cap[1].CanTx_config_request[0];
	Output.R1_10_ARR_CANrequest[1].data[1] := MCP_IO.MagDriver[1].Cap[1].CanTx_config_request[1];
	Output.R1_10_ARR_CANrequest[1].data[2] := MCP_IO.MagDriver[1].Cap[1].CanTx_config_request[2];
	Output.R1_10_ARR_CANrequest[1].data[3] := MCP_IO.MagDriver[1].Cap[1].CanTx_config_request[3];
	Output.R1_10_ARR_CANrequest[1].data[4] := MCP_IO.MagDriver[1].Cap[1].CanTx_config_request[4];
	Output.R1_10_ARR_CANrequest[1].data[5] := MCP_IO.MagDriver[1].Cap[1].CanTx_config_request[5];
	Output.R1_10_ARR_CANrequest[1].data[6] := MCP_IO.MagDriver[1].Cap[1].CanTx_config_request[6];
	Output.R1_10_ARR_CANrequest[1].data[7] := MCP_IO.MagDriver[1].Cap[1].CanTx_config_request[7];

	Output.R1_10_ARR_CANrequest[2].cobId := MCP_IO.MagDriver[1].Cap[2].CanTx_config_ID;
	Output.R1_10_ARR_CANrequest[2].data[0] := MCP_IO.MagDriver[1].Cap[2].CanTx_config_request[0];
	Output.R1_10_ARR_CANrequest[2].data[1] := MCP_IO.MagDriver[1].Cap[2].CanTx_config_request[1];
	Output.R1_10_ARR_CANrequest[2].data[2] := MCP_IO.MagDriver[1].Cap[2].CanTx_config_request[2];
	Output.R1_10_ARR_CANrequest[2].data[3] := MCP_IO.MagDriver[1].Cap[2].CanTx_config_request[3];
	Output.R1_10_ARR_CANrequest[2].data[4] := MCP_IO.MagDriver[1].Cap[2].CanTx_config_request[4];
	Output.R1_10_ARR_CANrequest[2].data[5] := MCP_IO.MagDriver[1].Cap[2].CanTx_config_request[5];
	Output.R1_10_ARR_CANrequest[2].data[6] := MCP_IO.MagDriver[1].Cap[2].CanTx_config_request[6];
	Output.R1_10_ARR_CANrequest[2].data[7] := MCP_IO.MagDriver[1].Cap[2].CanTx_config_request[7];
	
	// input
	
	//MCP_IO.MagDriver[1].Cap[1].Elec_AveVolt 		:= Input.R1_10_CapNumber[1].Status.Elec_AveVolt; //per cell <- example
	//this is replaced by the loop below
(*	MCP_IO.MagDriver[1].Cap[1].Elec_AveVolt 		:= Input.R1_10_CapNumber[1].Status.Elec_AveVolt; //per cell
	MCP_IO.MagDriver[1].Cap[1].Elec_Balancing 		:= Input.R1_10_CapNumber[1].Status.Elec_Balancing; // 0x0[Not Active], 0x1[Active], 0x2[Error], 0x3[Not Available]
	MCP_IO.MagDriver[1].Cap[1].Elec_HighestVolt 	:= Input.R1_10_CapNumber[1].Status.Elec_HighestVolt; //per cell
	MCP_IO.MagDriver[1].Cap[1].Elec_Imbalance 		:= Input.R1_10_CapNumber[1].Status.Elec_Imbalance;  // 0x0[No Warnings], 0x1[Warning Active], 0x2[Alarm Active], 0x3[Not Available]
	MCP_IO.MagDriver[1].Cap[1].Elec_OverVoltage		:= Input.R1_10_CapNumber[1].Status.Elec_OverVoltage;  // 0x0[No Warnings], 0x1[Warning Active], 0x2[Alarm Active], 0x3[NOT Available] 
	MCP_IO.MagDriver[1].Cap[1].Elec_VoltageSum		:= Input.R1_10_CapNumber[1].Status.Elec_VoltageSum; //total voltage in one UC
	MCP_IO.MagDriver[1].Cap[1].Therm_HighestCell	:= Input.R1_10_CapNumber[1].Status.Therm_HighestCell; //C
	MCP_IO.MagDriver[1].Cap[1].Therm_HighTemp		:= Input.R1_10_CapNumber[1].Status.Therm_HighTemp;  //0x0[No Warnings], 0x1[Warning Active], 0x2[Alarm Active], 0x3[NOT Available]
*)	
//need to verify the couunter
	FOR i := 1 TO n BY 1 DO 
		FOR j := 1 TO m BY 1 DO 
			IF j = 1 THEN 
				k := 2*i -j;
				ELSIF j = 2 THEN 
					k :=j*i;
			END_IF

			MCP_IO.MagDriver[i].Cap[j].Elec_AveVolt			:= Input.R1_10_CapNumber[k].Elec_AveVolt; //per cell
			MCP_IO.MagDriver[i].Cap[j].Elec_Balancing		:= Input.R1_10_CapNumber[k].Elec_Balancing; // 0x0[Not Active], 0x1[Active], 0x2[Error], 0x3[Not Available]
			MCP_IO.MagDriver[i].Cap[j].Elec_HighestVolt		:= Input.R1_10_CapNumber[k].Elec_HighestVolt; //per cell
			MCP_IO.MagDriver[i].Cap[j].Elec_Imbalance		:= Input.R1_10_CapNumber[k].Elec_Imbalance;  // 0x0[No Warnings], 0x1[Warning Active], 0x2[Alarm Active], 0x3[Not Available]
			MCP_IO.MagDriver[i].Cap[j].Elec_OverVoltage		:= Input.R1_10_CapNumber[k].Elec_OverVoltage;  // 0x0[No Warnings], 0x1[Warning Active], 0x2[Alarm Active], 0x3[NOT Available] 
			MCP_IO.MagDriver[i].Cap[j].Elec_VoltageSum		:= Input.R1_10_CapNumber[k].Elec_VoltageSum; //total voltage in one UC
			MCP_IO.MagDriver[i].Cap[j].Therm_HighestCell	:= Input.R1_10_CapNumber[k].Therm_HighestCell; //C
			MCP_IO.MagDriver[i].Cap[j].Therm_HighTemp		:= Input.R1_10_CapNumber[k].Therm_HighTemp;  //0x0[No Warnings], 0x1[Warning Active], 0x2[Alarm Active], 0x3[NOT Available]
			//uncomment to replace the code above - but only if we want to be able to edit ID on each and every single CAN ID
			(*Output.R1_10_ARR_CANrequest[i].data[0] := MCP_IO.MagDriver[i].Cap[k].CanTx_config_request[0];
			Output.R1_10_ARR_CANrequest[i].data[1] := MCP_IO.MagDriver[i].Cap[k].CanTx_config_request[1];
			Output.R1_10_ARR_CANrequest[i].data[2] := MCP_IO.MagDriver[i].Cap[k].CanTx_config_request[2];
			Output.R1_10_ARR_CANrequest[i].data[3] := MCP_IO.MagDriver[i].Cap[k].CanTx_config_request[3];
			Output.R1_10_ARR_CANrequest[i].data[4] := MCP_IO.MagDriver[i].Cap[k].CanTx_config_request[4];
			Output.R1_10_ARR_CANrequest[i].data[5] := MCP_IO.MagDriver[i].Cap[k].CanTx_config_request[5];
			Output.R1_10_ARR_CANrequest[i].data[6] := MCP_IO.MagDriver[i].Cap[k].CanTx_config_request[6];
			Output.R1_10_ARR_CANrequest[i].data[7] := MCP_IO.MagDriver[i].Cap[k].CanTx_config_request[7];*)
			MCP_IO.MagDriver[i].Cap[j].UltraCap_Dummy.R1_10_UC_Rx_cobID := Input.R1_10_UC_status[k].R1_10_UC_Rx_cobID;
			MCP_IO.MagDriver[i].Cap[j].UltraCap_Dummy.R1_10_UC_Rx_data := Input.R1_10_UC_status[k].R1_10_UC_Rx_data;
		END_FOR		
	END_FOR
	
	//MCP_IO.MagDriver[1].Cap[1].UltraCap_Dummy.R1_10_UC_Rx_cobID := Input.R1_10_UC_7F_status.R1_10_UC_Rx_cobID;
	//MCP_IO.MagDriver[1].Cap[1].UltraCap_Dummy.R1_10_UC_Rx_data := Input.R1_10_UC_7F_status.R1_10_UC_Rx_data;	
	// need to have how many voltage monitor board or voltage transmitter board per fruit stand ????
	//LCP3_IO.VMB.VTB[1].

	//LV Alias
	//commented out to test the sequence
(*	
	HMI_DB.ChargePB 				:= LV.TxWord1.0;
	HMI_DB.DumpPB					:= LV.TxWord1.1;		
	HMI_DB.AbortPB					:= LV.TxWord1.2;
	HMI_DB.FirePB					:= LV.TxWord1.3;
	HMI_DB.ClearFaultPB 			:= LV.TxWord1.4;
	HMI_DB.AllDumpRelaysOpenBP		:= LV.TxWord1.5;
	HMI_DB.AllChargeRelayCloseBP	:= LV.TxWord1.6;
	HMI_DB.SystemSafeBP				:= LV.TxWord1.7;
	HMI_DB.CloseChargeRlySW			:= LV.TxWord1.8;
	HMI_DB.OpenDumpRlySW 			:= LV.TxWord1.9;
	HMI_DB.HMI_ManualModeSelected	:= LV.TxWord1.10;  // 1 = manual mode selected
	HMI_DB.TurnChrgInhibitOffSW		:= LV.TxWord1.11;
	HMI_DB.TurnOnShotTrigSW			:= LV.TxWord1.12;
	HMI_DB.TurnOnChargeAlarm		:= LV.TxWord1.13;
	//:= LV.TxWord1.14;
	//:= LV.TxWord1.15;
	
	MCP_IO.Charger[1].inhibit		:= LV.TxWord2.0;
	MCP_IO.Charger[2].inhibit		:= LV.TxWord2.1;
	MCP_IO.Charger[3].inhibit		:= LV.TxWord2.2;
	MCP_IO.Charger[4].inhibit		:= LV.TxWord2.3;
	
	MCP_IO.Charger[5].inhibit		:= LV.TxWord2.4;
	MCP_IO.Charger[6].inhibit		:= LV.TxWord2.5;
	
	LV.RxWord1.0 := MCP_IO.MagDriver[1].SCR_ready_to_fire;
	LV.RxWord1.1 := MCP_IO.MagDriver[2].SCR_ready_to_fire;
	LV.RxWord1.2 := MCP_IO.MagDriver[3].SCR_ready_to_fire;
	LV.RxWord1.3 := MCP_IO.MagDriver[4].SCR_ready_to_fire;
	LV.RxWord1.4 := MCP_IO.MagDriver[5].SCR_ready_to_fire;
	LV.RxWord1.5 := MCP_IO.MagDriver[6].SCR_ready_to_fire;
	LV.RxWord1.6 := Permissives_DB.AllSCRreadyToFire;
	//LV.RxWord1.7 
	//LV.RxWord1.8 
	//LV.RxWord1.9 
	//LV.RxWord1.10
	//LV.RxWord1.11 
	//LV.RxWord1.12 
	//LV.RxWord1.13 
	//LV.RxWord1.14 
	//LV.RxWord1.15 
	
	LV.RxWord2.0 := MCP_IO.MagDriver[1].ChargeRelayClose;
	LV.RxWord2.1 := MCP_IO.MagDriver[2].ChargeRelayClose;
	LV.RxWord2.2 := MCP_IO.MagDriver[3].ChargeRelayClose;
	LV.RxWord2.3 := MCP_IO.MagDriver[4].ChargeRelayClose;
	LV.RxWord2.4 := MCP_IO.MagDriver[5].ChargeRelayClose;
	LV.RxWord2.5 := MCP_IO.MagDriver[6].ChargeRelayClose;
	LV.RxWord2.6 := Permissives_DB.AllChargeRelayClosed;
	LV.RxWord2.7 := MCP_IO.MagDriver[1].DumpRelayOpen;
	LV.RxWord2.8 := MCP_IO.MagDriver[2].DumpRelayOpen;
	LV.RxWord2.9 := MCP_IO.MagDriver[3].DumpRelayOpen;
	LV.RxWord2.10 := MCP_IO.MagDriver[4].DumpRelayOpen;
	LV.RxWord2.11 := MCP_IO.MagDriver[5].DumpRelayOpen;
	LV.RxWord2.12 := MCP_IO.MagDriver[6].DumpRelayOpen;
	LV.RxWord2.13 := Permissives_DB.AllDumpRelayOpen;
	LV.RxWord3.14 := Permissives_DB.AllDumpResTempOK;
	//LV.RxWord3.15   
	
	HMI_DB.ChargerHVOFF_rlyDelayPT_INT	:= LV.TxInt[1];
	HMI_DB.HVONdelayPT_INT 				:= LV.TxInt[2];
	LV.RxInt[1]							:= HMI_DB.ChargingRunOutTMR_elapse;
	
	HMI_DB.RunOutTMR_PT_INT				:= LV.TxDint[1];
	LV.RxDint[1]						:= HMI_DB.RunOutTMR_elapse;	
	
	FOR i := 1 TO n BY 1 DO
		
		HMI_DB.HPT5[i].RequiredChargedV				:= LV.HPT5Load[i].RequiredChargedV; // manually enter voltage setpoint
		//HMI_DB.HPT5[i].TotalCapacitance	:= LV.HPT5Load[i].TotalCapacitance;	
		HMI_DB.HPT5[i].ChargeTime					:= LV.HPT5Load[i].ChargeTime;	//manually enter charge time
		LV.Charger[i].ChargeTime.timeToChargeLoad 	:= MCP_IO.Charger[i].ChargeTime.timeToChargeLoad; //send charge time back to LV
		
	END_FOR
	 
	LV.RxREAL[1] := MCP_IO.MagDriver[1].Cap[1].CapVoltage; 
	LV.RxREAL[2] := MCP_IO.MagDriver[1].Cap[2].CapVoltage;  
	LV.RxREAL[3] := MCP_IO.MagDriver[2].Cap[1].CapVoltage;  
	LV.RxREAL[4] := MCP_IO.MagDriver[2].Cap[2].CapVoltage;  
	LV.RxREAL[5] := MCP_IO.MagDriver[3].Cap[1].CapVoltage;  
	LV.RxREAL[6] := MCP_IO.MagDriver[3].Cap[2].CapVoltage;  
	LV.RxREAL[7] := MCP_IO.MagDriver[4].Cap[1].CapVoltage;  
	LV.RxREAL[8] := MCP_IO.MagDriver[4].Cap[2].CapVoltage;  
	LV.RxREAL[9] := MCP_IO.MagDriver[5].Cap[1].CapVoltage;  
	LV.RxREAL[10] := MCP_IO.MagDriver[5].Cap[2].CapVoltage;  
	LV.RxREAL[11] := MCP_IO.MagDriver[6].Cap[1].CapVoltage;  
	LV.RxREAL[12] := MCP_IO.MagDriver[6].Cap[2].CapVoltage;   
	
	LV.RxREAL[13] := MCP_IO.MagDriver[1].DumpResistorTemp; 
	LV.RxREAL[14] := MCP_IO.MagDriver[2].DumpResistorTemp; 
	LV.RxREAL[15] := MCP_IO.MagDriver[3].DumpResistorTemp; 
	LV.RxREAL[16] := MCP_IO.MagDriver[4].DumpResistorTemp; 
	LV.RxREAL[17] := MCP_IO.MagDriver[5].DumpResistorTemp; 
	LV.RxREAL[18] := MCP_IO.MagDriver[6].DumpResistorTemp; 
	
	LV.ReadState 						:= Sequence.eState;	 
	plc_plc_comm_DB.ReadStateFromPLC 	:= LV.WriteState;
	LV.database 						:= P_TextModeWrite.database;
	*)
	

IF j > m THEN 
	j := 1;
END_IF

IF i > n THEN 
	i := 1;
END_IF

IF k > p THEN 
	k := 1;
END_IF

END_PROGRAM

// ---- POUs/CAN_comm.TcPOU
PROGRAM CAN_comm
VAR
	i : INT := 1; // mag driver 1 - 6
	n : INT := 6; //
	j : INT := 1; // cap 1 - 2
	m : INT := 2;

	hmi_sendRequest : BOOL;
	hmi_step1 : BOOL;
	hmi_step2 : BOOL;
	hmi_step3 : BOOL;
	hmi_step4 : BOOL;
	hmi_step5 : BOOL;
	//hmi_CanTxB_str	: ARRAY [0..7] OF STRING;
	//hmi_CanTxB		: ARRAY [0..7] OF BYTE;
	hmi_CanTx_ID_str	: STRING;
	hmi_CanTx_ID		: UDINT;
	//hmi_CanTx_length	: UINT;
	hmi_CanTx_desiredID : STRING;
	hmi_CanTx_desID		: BYTE;
	
	//hmi CanTx 7F only
	UC_7F_ID_hexstr		: STRING;
	hmi_CanTx_7F_ID_str	: STRING;
	hmi_CanTx_7F_ID		: UDINT;
	//hmi_CanTx_length	: UINT;
	hmi_CanTx_7F_desiredID : STRING;
	hmi_CanTx_7F_desID		: BYTE;
	
	hmi_7F_step1 : BOOL;
	hmi_7F_step2 : BOOL;
	hmi_7F_step3 : BOOL;
	hmi_7F_step4 : BOOL;
	hmi_7F_step5 : BOOL;
	
	CanTx_7F_config_ID 	: UDINT;
	CanTx_7F_config_length : UINT;
	CanTx_7F_config_request: ARRAY[0..7] OF BYTE;
END_VAR

//0x0CF091 XX ELECTRICAL DATA
//0x0CF092 XX THERMAL DATA

//XX 
// ie 0x11[overvoltage][imbalance][blancing]
//data[0] = Electrical flag | data[1], data[2] = Voltage sum | data[3], data[4] = highest voltage | data[5], data[6] = average voltage | data[7] = life counter
//data[0].0
//data[0].1  Balancing
//data[0].2  
//data[0].3  Imbalance
//data[0].4
//data[0].5  Overvoltage
//data[0].6 = 1
//data[0].7 = 1



	//Devices.Coil[1].UltraCap_CAN_ID := Replace (STR1 := Devices.Coil[1].UltraCap_CAN_ID, '',1,1);
	//Devices.Coil[j].UltraCap_CAN_RxMsgNum[k].cobID := LEFT (Devices.Coil[j].UltraCap_CAN_RxMsgNum[k].cobID, 5);

(*	Devices.Coil[j].UltraCap_CAN_RxMsgNum[0].byteData_hexstr[0] := BYTE_TO_HEXSTR (in := Devices.Coil[j].UltraCap_CAN_RxMsg[0].data[0], iPrecision := 2, bLoCase := FALSE);
	Devices.Coil[j].UltraCap_CAN_RxMsgNum[0].byteData_hexstr[1] := BYTE_TO_HEXSTR (in := Devices.Coil[j].UltraCap_CAN_RxMsg[0].data[1], iPrecision := 2, bLoCase := FALSE);
	Devices.Coil[j].UltraCap_CAN_RxMsgNum[0].byteData_hexstr[2] := BYTE_TO_HEXSTR (in := Devices.Coil[j].UltraCap_CAN_RxMsg[0].data[2], iPrecision := 2, bLoCase := FALSE);
	Devices.Coil[j].UltraCap_CAN_RxMsgNum[0].byteData_hexstr[3] := BYTE_TO_HEXSTR (in := Devices.Coil[j].UltraCap_CAN_RxMsg[0].data[3], iPrecision := 2, bLoCase := FALSE);
	Devices.Coil[j].UltraCap_CAN_RxMsgNum[0].byteData_hexstr[4] := BYTE_TO_HEXSTR (in := Devices.Coil[j].UltraCap_CAN_RxMsg[0].data[4], iPrecision := 2, bLoCase := FALSE);
	Devices.Coil[j].UltraCap_CAN_RxMsgNum[0].byteData_hexstr[5] := BYTE_TO_HEXSTR (in := Devices.Coil[j].UltraCap_CAN_RxMsg[0].data[5], iPrecision := 2, bLoCase := FALSE);
	Devices.Coil[j].UltraCap_CAN_RxMsgNum[0].byteData_hexstr[6] := BYTE_TO_HEXSTR (in := Devices.Coil[j].UltraCap_CAN_RxMsg[0].data[6], iPrecision := 2, bLoCase := FALSE);
	Devices.Coil[j].UltraCap_CAN_RxMsgNum[0].byteData_hexstr[7] := BYTE_TO_HEXSTR (in := Devices.Coil[j].UltraCap_CAN_RxMsg[0].data[7], iPrecision := 2, bLoCase := FALSE);
	*)
	
(* 	HOW TO USE THE CAN BUS ID EDIT FUNCTION
1. enter the cobID 	: 16#0CDA<xx>CC  <- this is the current Capacitor ID that you would like it to be different.
2. enter the Desired ID# : 16#yy  (01..FE)	<- this is the CAN ID that you would like the capacitor to be. Valid ID ranges from x01 to xFE
3. enter Mag Driver #: 1-6 	<- this is the mag driver number (rack number) that corresponds to the output address of the PLC that is mapped to send to the specific CAN ID.
4. enter the Cap #: 1-2		<- this is the capacitor number (cap 1 or cap 2) then corresponds to the output address of the PLC that is mapped to send to the specific CAN ID.

*there are total of 6 mag drivers, and each has 2 capacitors.

5. Press "Step1 Send", this should cue up the MSG ID of the Cap, and the Device ID of that cap will be shown
6. Press "Step2, Step3, Step4, and Step5" in a sequence.  <- this should change the CAN ID 

if a newly added Cap, the default ID is 7F.
The use the 7F section to set the ID to a unique ID.
*)
FOR i := 1 TO 6 BY 1 DO 	
	FOR j := 1 TO 2 BY 1 DO 
	 	//verify the counter
		MCP_IO.MagDriver[i].Cap[j].UC_Dummy_ID_hexstr :=  (DWORD_TO_HEXSTR (in := MCP_IO.MagDriver[i].Cap[j].UltraCap_Dummy.R1_10_UC_Rx_cobID, iPrecision := 2, bLoCase := FALSE));
		MCP_IO.MagDriver[i].Cap[j].CapVoltage := LREAL_TO_REAL (MCP_IO.MagDriver[i].Cap[j].Elec_VoltageSum);
		MCP_IO.MagDriver[i].Cap[j].CapCellTemp := LREAL_TO_REAL (MCP_IO.MagDriver[i].Cap[j].Therm_HighestCell); //sample the highest cell temperature
	
	END_FOR;
END_FOR;

// 01
MCP_IO.MagDriver[1].Cap[1].UC_Dummy_ID_hexstr :=  (DWORD_TO_HEXSTR (in := MCP_IO.MagDriver[1].Cap[1].UltraCap_Dummy.R1_10_UC_Rx_cobID, iPrecision := 2, bLoCase := FALSE));
// 7F
UC_7F_ID_hexstr := (DWORD_TO_HEXSTR (in := Input.R1_10_UC_7F_status.R1_10_UC_Rx_cobID, iPrecision := 2, bLoCase := FALSE));


//output set address for new UC - 01..FE 
//taking input from HMI
hmi_CanTx_ID := STRING_TO_UDINT (hmi_CanTx_ID_str);
hmi_CanTx_desID := STRING_TO_BYTE (hmi_CanTx_desiredID);

//output set address for new UC - 7F 
hmi_CanTx_7F_ID := STRING_TO_UDINT (hmi_CanTx_7F_ID_str);	
hmi_CanTx_7F_desID	:= STRING_TO_BYTE (hmi_CanTx_7F_desiredID);


(*FOR i := 0 TO 7 BY 1 DO 
	hmi_CanTxB[i] := STRING_TO_BYTE (hmi_CanTxB_str[i]);
END_FOR;
	
IF hmi_sendRequest = TRUE THEN
	Devices.Coil[1].CanTx_config_ID := hmi_CanTx_ID;
	Devices.Coil[1].CanTx_config_length := hmi_CanTx_length;
	Devices.Coil[1].CanTx_config_request[0] := hmi_CanTxB[0];
	Devices.Coil[1].CanTx_config_request[1] := hmi_CanTxB[1];
	Devices.Coil[1].CanTx_config_request[2] := hmi_CanTxB[2];
	Devices.Coil[1].CanTx_config_request[3] := hmi_CanTxB[3];
	Devices.Coil[1].CanTx_config_request[4] := hmi_CanTxB[4];
ELSE 
	Devices.Coil[1].CanTx_config_ID := 16#00000000;
	Devices.Coil[1].CanTx_config_request[0] := 16#00;
	Devices.Coil[1].CanTx_config_request[1] := 16#00;
	Devices.Coil[1].CanTx_config_request[2] := 16#00;
	Devices.Coil[1].CanTx_config_request[3] := 16#00;
	Devices.Coil[1].CanTx_config_request[4] := 16#00;
	Devices.Coil[1].CanTx_config_request[5] := 16#00;
	Devices.Coil[1].CanTx_config_request[6] := 16#00;
	Devices.Coil[1].CanTx_config_request[7] := 16#00;
END_IF;
*)
//limits
IF HMI_DB.CAN_Comm_MagDriverNum > 6 THEN 
	HMI_DB.CAN_Comm_MagDriverNum := 6;
ELSIF  HMI_DB.CAN_Comm_MagDriverNum < 0 THEN 
	HMI_DB.CAN_Comm_MagDriverNum := 0;
END_IF
IF HMI_DB.CAN_Comm_UC_Num > 2 THEN 
	HMI_DB.CAN_Comm_UC_Num := 2;
ELSIF  HMI_DB.CAN_Comm_UC_Num < 0 THEN 
	HMI_DB.CAN_Comm_UC_Num := 0;
END_IF

IF hmi_step1 = TRUE THEN
	(*MCP_IO.MagDriver[1].Cap[1].CanTx_config_ID 			:= hmi_CanTx_ID;
	MCP_IO.MagDriver[1].Cap[1].CanTx_config_length 		:= 3;
	MCP_IO.MagDriver[1].Cap[1].CanTx_config_request[0] 	:= 16#02;
	MCP_IO.MagDriver[1].Cap[1].CanTx_config_request[1] 	:= 16#10;
	MCP_IO.MagDriver[1].Cap[1].CanTx_config_request[2] 	:= 16#03;*)
	MCP_IO.MagDriver[HMI_DB.CAN_Comm_MagDriverNum].Cap[HMI_DB.CAN_Comm_UC_Num].CanTx_config_ID 			:= hmi_CanTx_ID;
	MCP_IO.MagDriver[HMI_DB.CAN_Comm_MagDriverNum].Cap[HMI_DB.CAN_Comm_UC_Num].CanTx_config_length 		:= 3;
	MCP_IO.MagDriver[HMI_DB.CAN_Comm_MagDriverNum].Cap[HMI_DB.CAN_Comm_UC_Num].CanTx_config_request[0] 	:= 16#02;
	MCP_IO.MagDriver[HMI_DB.CAN_Comm_MagDriverNum].Cap[HMI_DB.CAN_Comm_UC_Num].CanTx_config_request[1] 	:= 16#10;
	MCP_IO.MagDriver[HMI_DB.CAN_Comm_MagDriverNum].Cap[HMI_DB.CAN_Comm_UC_Num].CanTx_config_request[2] 	:= 16#03;
	// add cap 2 - 6 
	
(*	Output.R2_06_CANrequest.cobId := 16#0CDA7FCC;
	Output.R2_06_CANrequest.length := 3;
	Output.R2_06_CANrequest.data[0] := 16#02;
	Output.R2_06_CANrequest.data[1] := 16#10;
	Output.R2_06_CANrequest.data[2] := 16#03;
	Output.R2_06_CANrequest.data[3] := 16#00;
	Output.R2_06_CANrequest.data[4] := 16#00;
	Output.R2_06_CANrequest.data[5] := 16#00;
	Output.R2_06_CANrequest.data[6] := 16#00;
	Output.R2_06_CANrequest.data[7] := 16#00;*)

ELSIF hmi_step2 = TRUE THEN
	(*MCP_IO.MagDriver[1].Cap[1].CanTx_config_ID := hmi_CanTx_ID;
	MCP_IO.MagDriver[1].Cap[1].CanTx_config_length := 3;
	MCP_IO.MagDriver[1].Cap[1].CanTx_config_request[0] := 16#02;
	MCP_IO.MagDriver[1].Cap[1].CanTx_config_request[1] := 16#27;
	MCP_IO.MagDriver[1].Cap[1].CanTx_config_request[2] := 16#03;*)
	
	MCP_IO.MagDriver[HMI_DB.CAN_Comm_MagDriverNum].Cap[HMI_DB.CAN_Comm_UC_Num].CanTx_config_ID := hmi_CanTx_ID;
	MCP_IO.MagDriver[HMI_DB.CAN_Comm_MagDriverNum].Cap[HMI_DB.CAN_Comm_UC_Num].CanTx_config_length := 3;
	MCP_IO.MagDriver[HMI_DB.CAN_Comm_MagDriverNum].Cap[HMI_DB.CAN_Comm_UC_Num].CanTx_config_request[0] := 16#02;
	MCP_IO.MagDriver[HMI_DB.CAN_Comm_MagDriverNum].Cap[HMI_DB.CAN_Comm_UC_Num].CanTx_config_request[1] := 16#27;
	MCP_IO.MagDriver[HMI_DB.CAN_Comm_MagDriverNum].Cap[HMI_DB.CAN_Comm_UC_Num].CanTx_config_request[2] := 16#03;
	(*Output.R2_06_CANrequest.cobId := 16#0CDA7FCC;
	Output.R2_06_CANrequest.length := 3;
	Output.R2_06_CANrequest.data[0] := 16#02;
	Output.R2_06_CANrequest.data[1] := 16#27;
	Output.R2_06_CANrequest.data[2] := 16#01;
	Output.R2_06_CANrequest.data[3] := 16#00;
	Output.R2_06_CANrequest.data[4] := 16#00;
	Output.R2_06_CANrequest.data[5] := 16#00;
	Output.R2_06_CANrequest.data[6] := 16#00;
	Output.R2_06_CANrequest.data[7] := 16#00;
	*)
ELSIF hmi_step3 = TRUE THEN
	(*MCP_IO.MagDriver[1].Cap[1].CanTx_config_ID := hmi_CanTx_ID;
	MCP_IO.MagDriver[1].Cap[1].CanTx_config_length := 5;
	MCP_IO.MagDriver[1].Cap[1].CanTx_config_request[0] := 16#04;
	MCP_IO.MagDriver[1].Cap[1].CanTx_config_request[1] := 16#27;
	MCP_IO.MagDriver[1].Cap[1].CanTx_config_request[2] := 16#02;
	MCP_IO.MagDriver[1].Cap[1].CanTx_config_request[3] := 16#78;
	MCP_IO.MagDriver[1].Cap[1].CanTx_config_request[4] := 16#9A;*)
	MCP_IO.MagDriver[HMI_DB.CAN_Comm_MagDriverNum].Cap[HMI_DB.CAN_Comm_UC_Num].CanTx_config_ID := hmi_CanTx_ID;
	MCP_IO.MagDriver[HMI_DB.CAN_Comm_MagDriverNum].Cap[HMI_DB.CAN_Comm_UC_Num].CanTx_config_length := 5;
	MCP_IO.MagDriver[HMI_DB.CAN_Comm_MagDriverNum].Cap[HMI_DB.CAN_Comm_UC_Num].CanTx_config_request[0] := 16#04;
	MCP_IO.MagDriver[HMI_DB.CAN_Comm_MagDriverNum].Cap[HMI_DB.CAN_Comm_UC_Num].CanTx_config_request[1] := 16#27;
	MCP_IO.MagDriver[HMI_DB.CAN_Comm_MagDriverNum].Cap[HMI_DB.CAN_Comm_UC_Num].CanTx_config_request[2] := 16#02;
	MCP_IO.MagDriver[HMI_DB.CAN_Comm_MagDriverNum].Cap[HMI_DB.CAN_Comm_UC_Num].CanTx_config_request[3] := 16#78;
	MCP_IO.MagDriver[HMI_DB.CAN_Comm_MagDriverNum].Cap[HMI_DB.CAN_Comm_UC_Num].CanTx_config_request[4] := 16#9A;
	(*Output.R2_06_CANrequest.cobId := 16#0CDA7FCC;
	Output.R2_06_CANrequest.length := 5;
	Output.R2_06_CANrequest.data[0] := 16#04;
	Output.R2_06_CANrequest.data[1] := 16#27;
	Output.R2_06_CANrequest.data[2] := 16#02;
	Output.R2_06_CANrequest.data[3] := 16#78;
	Output.R2_06_CANrequest.data[4] := 16#9A;
	Output.R2_06_CANrequest.data[5] := 16#00;
	Output.R2_06_CANrequest.data[6] := 16#00;
	Output.R2_06_CANrequest.data[7] := 16#00;	
	*)
ELSIF hmi_step4 = TRUE THEN 
	MCP_IO.MagDriver[HMI_DB.CAN_Comm_MagDriverNum].Cap[HMI_DB.CAN_Comm_UC_Num].CanTx_config_ID := hmi_CanTx_ID;
	MCP_IO.MagDriver[HMI_DB.CAN_Comm_MagDriverNum].Cap[HMI_DB.CAN_Comm_UC_Num].CanTx_config_length := 5;
	MCP_IO.MagDriver[HMI_DB.CAN_Comm_MagDriverNum].Cap[HMI_DB.CAN_Comm_UC_Num].CanTx_config_request[0] := 16#04;
	MCP_IO.MagDriver[HMI_DB.CAN_Comm_MagDriverNum].Cap[HMI_DB.CAN_Comm_UC_Num].CanTx_config_request[1] := 16#2E;
	MCP_IO.MagDriver[HMI_DB.CAN_Comm_MagDriverNum].Cap[HMI_DB.CAN_Comm_UC_Num].CanTx_config_request[2] := 16#FD;
	MCP_IO.MagDriver[HMI_DB.CAN_Comm_MagDriverNum].Cap[HMI_DB.CAN_Comm_UC_Num].CanTx_config_request[3] := 16#08;
	MCP_IO.MagDriver[HMI_DB.CAN_Comm_MagDriverNum].Cap[HMI_DB.CAN_Comm_UC_Num].CanTx_config_request[4] := hmi_CanTx_desID; //desirable cobID / device ID
	(*Output.R2_06_CANrequest.cobId := 16#0CDA7FCC;
	Output.R2_06_CANrequest.length := 5;
	Output.R2_06_CANrequest.data[0] := 16#04;
	Output.R2_06_CANrequest.data[1] := 16#2E;
	Output.R2_06_CANrequest.data[2] := 16#FD;
	Output.R2_06_CANrequest.data[3] := 16#08;
	Output.R2_06_CANrequest.data[4] := 16#02; //desirable cobID / device ID
	Output.R2_06_CANrequest.data[5] := 16#00;
	Output.R2_06_CANrequest.data[6] := 16#00;
	Output.R2_06_CANrequest.data[7] := 16#00;
	*)
ELSIF hmi_step5 = TRUE THEN 
	(*MCP_IO.MagDriver[1].Cap[1].CanTx_config_ID := hmi_CanTx_ID;
	MCP_IO.MagDriver[1].Cap[1].CanTx_config_length := 4;
	MCP_IO.MagDriver[1].Cap[1].CanTx_config_request[0] := 16#03; //restart software
	MCP_IO.MagDriver[1].Cap[1].CanTx_config_request[1] := 16#11;
	MCP_IO.MagDriver[1].Cap[1].CanTx_config_request[2] := 16#01;
	MCP_IO.MagDriver[1].Cap[1].CanTx_config_request[3] := 16#08;*)
	MCP_IO.MagDriver[HMI_DB.CAN_Comm_MagDriverNum].Cap[HMI_DB.CAN_Comm_UC_Num].CanTx_config_ID := hmi_CanTx_ID;
	MCP_IO.MagDriver[HMI_DB.CAN_Comm_MagDriverNum].Cap[HMI_DB.CAN_Comm_UC_Num].CanTx_config_length := 4;
	MCP_IO.MagDriver[HMI_DB.CAN_Comm_MagDriverNum].Cap[HMI_DB.CAN_Comm_UC_Num].CanTx_config_request[0] := 16#03; //restart software
	MCP_IO.MagDriver[HMI_DB.CAN_Comm_MagDriverNum].Cap[HMI_DB.CAN_Comm_UC_Num].CanTx_config_request[1] := 16#11;
	MCP_IO.MagDriver[HMI_DB.CAN_Comm_MagDriverNum].Cap[HMI_DB.CAN_Comm_UC_Num].CanTx_config_request[2] := 16#01;
	MCP_IO.MagDriver[HMI_DB.CAN_Comm_MagDriverNum].Cap[HMI_DB.CAN_Comm_UC_Num].CanTx_config_request[3] := 16#08;
	(*Output.R2_06_CANrequest.cobId:= 16#0CDA7FCC;
	Output.R2_06_CANrequest.length := 4;
	Output.R2_06_CANrequest.data[0] := 16#03;
	Output.R2_06_CANrequest.data[1] := 16#11;
	Output.R2_06_CANrequest.data[2] := 16#01;
	Output.R2_06_CANrequest.data[3] := 16#00;
	Output.R2_06_CANrequest.data[4] := 16#00;
	Output.R2_06_CANrequest.data[5] := 16#00;
	Output.R2_06_CANrequest.data[6] := 16#00;
	Output.R2_06_CANrequest.data[7] := 16#00;
	*)
ELSE 
	(*
	MCP_IO.MagDriver[1].Cap[1].CanTx_config_ID := 16#00000000;
	MCP_IO.MagDriver[1].Cap[1].CanTx_config_request[0] := 16#00;
	MCP_IO.MagDriver[1].Cap[1].CanTx_config_request[1] := 16#00;
	MCP_IO.MagDriver[1].Cap[1].CanTx_config_request[2] := 16#00;
	MCP_IO.MagDriver[1].Cap[1].CanTx_config_request[3] := 16#00;
	MCP_IO.MagDriver[1].Cap[1].CanTx_config_request[4] := 16#00;
	MCP_IO.MagDriver[1].Cap[1].CanTx_config_request[5] := 16#00;
	MCP_IO.MagDriver[1].Cap[1].CanTx_config_request[6] := 16#00;
	MCP_IO.MagDriver[1].Cap[1].CanTx_config_request[7] := 16#00;*)
	MCP_IO.MagDriver[HMI_DB.CAN_Comm_MagDriverNum].Cap[HMI_DB.CAN_Comm_UC_Num].CanTx_config_ID := 16#00000000;
	MCP_IO.MagDriver[HMI_DB.CAN_Comm_MagDriverNum].Cap[HMI_DB.CAN_Comm_UC_Num].CanTx_config_request[0] := 16#00;
	MCP_IO.MagDriver[HMI_DB.CAN_Comm_MagDriverNum].Cap[HMI_DB.CAN_Comm_UC_Num].CanTx_config_request[1] := 16#00;
	MCP_IO.MagDriver[HMI_DB.CAN_Comm_MagDriverNum].Cap[HMI_DB.CAN_Comm_UC_Num].CanTx_config_request[2] := 16#00;
	MCP_IO.MagDriver[HMI_DB.CAN_Comm_MagDriverNum].Cap[HMI_DB.CAN_Comm_UC_Num].CanTx_config_request[3] := 16#00;
	MCP_IO.MagDriver[HMI_DB.CAN_Comm_MagDriverNum].Cap[HMI_DB.CAN_Comm_UC_Num].CanTx_config_request[4] := 16#00;
	MCP_IO.MagDriver[HMI_DB.CAN_Comm_MagDriverNum].Cap[HMI_DB.CAN_Comm_UC_Num].CanTx_config_request[5] := 16#00;
	MCP_IO.MagDriver[HMI_DB.CAN_Comm_MagDriverNum].Cap[HMI_DB.CAN_Comm_UC_Num].CanTx_config_request[6] := 16#00;
	MCP_IO.MagDriver[HMI_DB.CAN_Comm_MagDriverNum].Cap[HMI_DB.CAN_Comm_UC_Num].CanTx_config_request[7] := 16#00;
	
END_IF;

// for 7F only ******************************  make a state machine for this later
IF hmi_7F_step1 = TRUE THEN
	CanTx_7F_config_ID 			:= hmi_CanTx_7F_ID;
	CanTx_7F_config_length 		:= 3;
	CanTx_7F_config_request[0] 	:= 16#02;
	CanTx_7F_config_request[1] 	:= 16#10;
	CanTx_7F_config_request[2] 	:= 16#03;
	
ELSIF hmi_7F_step2 = TRUE THEN
	CanTx_7F_config_ID := hmi_CanTx_7F_ID;
	CanTx_7F_config_length := 3;
	CanTx_7F_config_request[0] := 16#02;
	CanTx_7F_config_request[1] := 16#27;
	CanTx_7F_config_request[2] := 16#03;

ELSIF hmi_7F_step3 = TRUE THEN
	CanTx_7F_config_ID := hmi_CanTx_7F_ID;
	CanTx_7F_config_length := 5;
	CanTx_7F_config_request[0] := 16#04;
	CanTx_7F_config_request[1] := 16#27;
	CanTx_7F_config_request[2] := 16#02;
	CanTx_7F_config_request[3] := 16#78;
	CanTx_7F_config_request[4] := 16#9A;

ELSIF hmi_7F_step4 = TRUE THEN 
	CanTx_7F_config_ID := hmi_CanTx_7F_ID;
	CanTx_7F_config_length := 5;
	CanTx_7F_config_request[0] := 16#04;
	CanTx_7F_config_request[1] := 16#2E;
	CanTx_7F_config_request[2] := 16#FD;
	CanTx_7F_config_request[3] := 16#08;
	CanTx_7F_config_request[4] := hmi_CanTx_7F_desID; //desirable cobID / device ID

ELSIF hmi_7F_step5 = TRUE THEN 
	CanTx_7F_config_ID := hmi_CanTx_7F_ID;
	CanTx_7F_config_length := 4;
	CanTx_7F_config_request[0] := 16#03; //restart software
	CanTx_7F_config_request[1] := 16#11;
	CanTx_7F_config_request[2] := 16#01;
	CanTx_7F_config_request[3] := 16#08;

ELSE 
	CanTx_7F_config_ID  := 16#00000000;
	CanTx_7F_config_request[0] := 16#00;
	CanTx_7F_config_request[1] := 16#00;
	CanTx_7F_config_request[2] := 16#00;
	CanTx_7F_config_request[3] := 16#00;
	CanTx_7F_config_request[4] := 16#00;
	CanTx_7F_config_request[5] := 16#00;
	CanTx_7F_config_request[6] := 16#00;
	CanTx_7F_config_request[7] := 16#00;
	
END_IF;



//invalid volt and temp 
FOR i := 1 TO 6 BY 1 DO 	
	FOR j := 1 TO 2 BY 1 DO 
	 	IF MCP_IO.MagDriver[i].Cap[j].CapVoltage >= 327 THEN 
			//invalid 
			MCP_IO.MagDriver[i].Cap[j].CapVoltage := -null;
		END_IF
		IF MCP_IO.MagDriver[i].Cap[j].CapCellTemp >= 210 THEN 
	 		MCP_IO.MagDriver[i].Cap[j].CapCellTemp := -null;
		END_IF
	END_FOR;
END_FOR;



IF i > n THEN
	i := 1;
END_IF;

IF j > m THEN
	j := 1;
END_IF;

END_PROGRAM

// ---- POUs/csv/P_ArgToConvExample.TcPOU
PROGRAM P_ArgToConvExample
VAR
	(* PLC data to be converted to or from CSV format *)
	bOperating	: BOOL := TRUE;
	fAxPos		: LREAL := 12.2;
	nCounter 	: UDINT := 7;
	sName		: T_MaxString := 'Module: "XAF", $04$05, 20';
	binData		: ARRAY[0..9] OF BYTE :=[ 0, 1, 2, 3, 4, 5, 6, 7, 8, 9];
	sShort		: STRING(10) := 'XAF';

	(* conversion buffer *)
	field1 : ARRAY[0..50 ] OF BYTE;
	field2 : ARRAY[0..50 ] OF BYTE;
	field3 : ARRAY[0..50 ] OF BYTE;
	field4 : ARRAY[0..50 ] OF BYTE;
	field5 : ARRAY[0..50 ] OF BYTE;
	field6 : ARRAY[0..50 ] OF BYTE;

	cbField1 : UDINT;
	cbField2 : UDINT;
	cbField3 : UDINT;
	cbField4 : UDINT;
	cbField5 : UDINT;
	cbField6 : UDINT;

	cbVar1 : UDINT;
	cbVar2 : UDINT;
	cbVar3 : UDINT;
	cbVar4 : UDINT;
	cbVar5 : UDINT;
	cbVar6 : UDINT;

END_VAR

cbField1 := ARG_TO_CSVFIELD( F_BOOL( bOperating ), TRUE, ADR( field1 ), SIZEOF( field1 ) );
cbField2 := ARG_TO_CSVFIELD( F_LREAL( fAxPos ), TRUE, ADR( field2 ), SIZEOF( field2 ) );
cbField3 := ARG_TO_CSVFIELD( F_UDINT( nCounter ), TRUE, ADR( field3 ), SIZEOF( field3 ) );
cbField4 := ARG_TO_CSVFIELD( F_STRING( sName ), TRUE, ADR( field4 ), SIZEOF( field4 ) );
cbField5 := ARG_TO_CSVFIELD( F_BIGTYPE( ADR( binData ), SIZEOF( binData ) ), TRUE, ADR( field5 ), SIZEOF( field5 ) );
cbField6 := ARG_TO_CSVFIELD( F_BIGTYPE( ADR( sShort ), INT_TO_DWORD( LEN( sShort ) ) ), TRUE, ADR( field6 ), SIZEOF( field6 ) );

cbVar1 := CSVFIELD_TO_ARG( ADR( field1 ), cbField1, TRUE, F_BOOL( bOperating ) );
cbVar2 := CSVFIELD_TO_ARG( ADR( field2 ), cbField2, TRUE, F_LREAL( fAxPos ) );
cbVar3 := CSVFIELD_TO_ARG( ADR( field3 ), cbField3, TRUE, F_UDINT( nCounter ) );
cbVar4 := CSVFIELD_TO_ARG( ADR( field4 ), cbField4, TRUE, F_STRING( sName ) );
cbVar5 := CSVFIELD_TO_ARG( ADR( field5 ), cbField5, TRUE, F_BIGTYPE( ADR( binData ), SIZEOF( binData ) ) );
cbVar6 := CSVFIELD_TO_ARG( ADR( field6 ), cbField6, TRUE, F_BIGTYPE( ADR( sShort ), INT_TO_DWORD( LEN( sShort ) ) ) );

END_PROGRAM

// ---- POUs/csv/P_StringToConvExample.TcPOU
PROGRAM P_StringToConvExample
VAR
	s1	: STRING;
	s2	: STRING;
END_VAR

s1 := STRING_TO_CSVFIELD( 'Module_"ALFA_$05"_6', TRUE  );
s2 := STRING_TO_CSVFIELD( 'Module_50', FALSE );

s1 := CSVFIELD_TO_STRING( '"ab_$04_$05_cd-""ALFA""_5"', TRUE  );
s2 := CSVFIELD_TO_STRING( 'Module_50', FALSE );

END_PROGRAM

// ---- POUs/csv/P_TextModeRead.TcPOU
(* Reading of CSV file in text mode. None of the field value is containing any non-printing control characters like line feed, carriage return, quotation marks, semicolon... *)
PROGRAM P_TextModeRead
VAR
	bRead			: BOOL := FALSE;(* Rising edge starts program execution *)
	sNetId			: T_AmsNetId := '';	(* TwinCAT system network address *)
	sFileName		: T_MaxString := 'C:\CSVdata\TextModeGen.csv';(* CSV source file path and name *)
	sCSVLine		: T_MaxString := '';(* Single CSV text line (row, record), we are using string as record buffer (your are able to see read fields)  *)
	sCSVField		: T_MaxString := '';(* Single CSV field value (column, record field) *)
	bBusy			: BOOL;
	bError			: BOOL;
	nErrId			: UDINT;
	nRow	 		: UDINT 	:= 0;(* Row number (record) *)
	nColumn			: UDINT 	:= 0;(* Column number (record field) *)
	hFile			: UINT		:= 0;(* File handle of the source file *)
	step			: DWORD 	:= 0;
	fbFileOpen		: FB_FileOpen;(* Opens file *)
	fbFileClose		: FB_FileClose;(* Closes file *)
	fbFileGets		: FB_FileGets;(* Reads one record (line) *)
	fbReader		: FB_CSVMemBufferReader;(* Helper function block used to parse CSV data bytes (single record line) *)

	database		: ARRAY[0..plc_plc_comm_DB.MAX_CSV_ROWS, 0..plc_plc_comm_DB.MAX_CSV_COLUMNS ] OF STRING(plc_plc_comm_DB.MAX_CSV_FIELD_LENGTH);(* Target PLC database *)
END_VAR

CASE step OF
	0:	(* Wait for rising edge at bRead variable *)
		IF bRead THEN
			bRead 	:= FALSE;
			bBusy 	:= TRUE;
			bError	:= FALSE;
			nErrId	:= 0;
			hFile	:= 0;
			nRow	:= 0;
			nColumn	:= 0;
			MEMSET( ADR( database ), 0, SIZEOF( database ) );
			step 		:= 1;
		END_IF

	1:	(* Open source file *)
		fbFileOpen(  bExecute := FALSE  );
		fbFileOpen( sNetId := sNetId, sPathName := sFileName, nMode := FOPEN_MODEREAD OR FOPEN_MODETEXT,(* Open file in TEXT mode! *)
					ePath := PATH_GENERIC, bExecute := TRUE );
		step := 2;

	2:(* Wait until open not busy *)
		fbFileOpen( bExecute := FALSE, bError => bError, nErrID => nErrID, hFile => hFile );
		IF NOT fbFileOpen.bBusy THEN
			IF NOT fbFileOpen.bError THEN
				step := 3;
			ELSE(* Error: file not found? *)
				step := 100;
			END_IF
		END_IF

	3:	(* Read single line (record) *)
		fbFileGets( bExecute := FALSE );
		fbFileGets( sNetId := sNetId, hFile := hFile, bExecute := TRUE );
		step := 4;

	4:(* Wait until read not busy *)
		fbFileGets( bExecute := FALSE, bError => bError, nErrID => nErrID, sLine => sCSVLine );
		IF NOT fbFileGets.bBusy THEN
			IF NOT fbFileGets.bError THEN
				IF fbFileGets.bEOF THEN
					step := 10;(* End of file reached => Close source file *)
				ELSE

					(* FB_FileGets returns text line without the CR (carriage return) character.
					We have to restore the CR character (replace the $L character with $R$L characters) *)
					IF RIGHT( sCSVLine, 1 ) = '$L' THEN
						sCSVLine := REPLACE( sCSVLine, '$R$L', 2, LEN( sCSVLine ) );
					END_IF

					step := 5;
				END_IF
			ELSE(* Error *)
				step := 100;
			END_IF
		END_IF

	5:(* Parse single line (record) *)
		fbReader.eCmd := eEnumCmd_First;(* Read first field value *)
		REPEAT
			fbReader( pBuffer := ADR( sCSVLine ), cbBuffer := SIZEOF( sCSVLine ), getValue => sCSVField );
			IF fbReader.bOk THEN
				fbReader.eCmd := eEnumCmd_Next;(* Read next field value *)

				IF ( nRow <= plc_plc_comm_DB.MAX_CSV_ROWS ) THEN
					IF ( nColumn <= plc_plc_comm_DB.MAX_CSV_COLUMNS ) THEN
						database[nRow, nColumn] := CSVFIELD_TO_STRING( sCSVField, FALSE );(* TODO: Save or use the field value in your application *)
					END_IF
				END_IF

				nColumn := nColumn + 1;(* Increment number of read columns *)
				IF fbReader.bCRLF THEN(* CRLF == TRUE => End of reacord reached *)
					nRow 		:= nRow + 1;(* Increment number of read records *)
					nColumn 	:= 0;(* Reset number of columns *)
				END_IF

			ELSE(* Error: End of record reached or all fields read *)
				step := 3;(* Try to read next line *)
			END_IF
		UNTIL NOT fbReader.bOk
		END_REPEAT

	10:	(* Close source file *)
		fbFileClose( bExecute := FALSE );
		fbFileClose( sNetId := sNetId, hFile := hFile, bExecute := TRUE );
		step := 11;

	11:(* Wait until close not busy *)
		fbFileClose( bExecute := FALSE, bError => bError, nErrID => nErrID );
		IF ( NOT fbFileClose.bBusy ) THEN
			hFile := 0;
			step := 100;
		END_IF

	100: (* Error or ready step => cleanup *)
		IF ( hFile <> 0 ) THEN
			step := 10; (* Close the source file *)
		ELSE
			bBusy := FALSE;
			step := 0;	(* Ready *)
		END_IF

END_CASE

END_PROGRAM

// ---- POUs/csv/P_TextModeWrite.TcPOU
(* Writing of CSV file in text mode. None of the field value is containing any non-printing control characters like line feed, carriage return, quotation marks, semicolon... *)
PROGRAM P_TextModeWrite
VAR_INPUT
	bWrite			: BOOL := FALSE;(* Rising edge starts program execution *)
END_VAR
VAR
	//bWrite			: BOOL := FALSE;(* Rising edge starts program execution *)
	timer_TON		: TON;
	timer_PT		: TIME;
	timer_ET		: TIME;
	timestamp		: REAL;
	SysCLK			: GETSYSTEMTIME;
	fileTime		: T_FILETIME;
	location		: T_MaxString := 'C:\CSVdata\';
	fileType		: T_MaxString := '.csv';
	filename		: STRING;
	filename_full	: T_MaxString;
	filename_short	: T_MaxString;
	sNetId			: T_AmsNetId := '';	(* TwinCAT system network address *)
	sFileName		: T_MaxString := 'C:\CSVdata\ShotClog.csv';(* CSV destination file path and name *)
	sCSVLine		: T_MaxString := '';(* Single CSV text line (row, record), we are using string as record buffer (your are able to see created fields) *)
	sCSVField		: T_MaxString := '';(* Single CSV field value (column, record field) *)
	bBusy			: BOOL;
	bError			: BOOL;
	nErrId			: UDINT;
	nRow	 		: UDINT 	:= 0;(* Row number (record) *)
	nColumn			: UDINT 	:= 0;(* Column number (record field) *)
	hFile			: UINT		:= 0;(* File handle of the source file *)
	step			: DWORD 	:= 0;
	fbFileOpen		: FB_FileOpen;(* Opens file *)
	fbFileClose		: FB_FileClose;(* Closes file *)
	fbFilePuts		: FB_FilePuts;(* Writes one record (line) *)
	fbWriter		: FB_CSVMemBufferWriter;(* Helper function block used to create CSV data bytes (single record line) *)
	
	//eState 					: E_State;
	csvW_RebounceTMR_TON	: TON;
	csvW_RebounceTMR_PT		: TIME := T#500MS;
	StartLogging_ONS		: BOOL;
	i 						: UDINT := 0;
	SamplingTMR_TON 		: TON;
	SamplingTMR_PT			: TIME := T#1S;
	SamplingTMR_ET			: TIME;
	SaveCSV					: BOOL := FALSE;
	SaveBuff			: BOOL := FALSE;
	
	database		: ARRAY[0..GVL.MAX_CSV_ROWS, 0..GVL.MAX_CSV_COLUMNS ] OF STRING(GVL.MAX_CSV_FIELD_LENGTH) :=[ (* Source PLC database *)
	'0_0', '0_1', '0_2', '0_3', '0_4', '0_5', '0_6',
	'1_0', '1_1', '1_2', '1_3', '1_4', '1_5', '1_6',
	'2_0', '2_1', '2_2', '2_3', '2_4', '2_5', '2_6',
	'3_0', '3_1', '3_2', '3_3', '3_4', '3_5', '3_6',
	'4_0', '4_1', '4_2', '4_3', '4_4', '4_5', '4_6',
	'5_0', '5_1', '5_2', '5_3', '5_4', '5_5', '5_6'];
	


END_VAR

//add cap voltage or shot current here.

SysCLK (timeLoDW => fileTime.dwLowDateTime, timeHiDW => fileTime.dwHighDateTime);

filename_full := DT_TO_STRING (FILETIME_TO_DT (fileTIME));

//filename_short := DELETE (DELETE (RIGHT (filename_full, 19), 1, 14), 1, 16);// LEFT (STR := filename, 35);
//sFileName := CONCAT (STR1 := 'C:\CSVdata\', STR2 := filename);
//filename := CONCAT (STR1 := filename_short, STR2 := fileType); //incrementing file name
//sFileName := CONCAT (STR1 := location, STR2 := filename);
CASE step OF
	0:	(* Wait for rising edge at bWrite variable *)
		IF bWrite THEN
			bWrite 	:= FALSE;
			bBusy 	:= TRUE;
			bError	:= FALSE;
			nErrId	:= 0;
			hFile	:= 0;
			nRow	:= 0;
			nColumn	:= 0;
			step 	:= 1;
		END_IF

	1:	(* Open source file *)
		fbFileOpen(  bExecute := FALSE  );
		
		filename_short := DELETE (DELETE (RIGHT (filename_full, 19), 1, 14), 1, 16);// LEFT (STR := filename, 35);
		filename := CONCAT (STR1 := filename_short, STR2 := fileType); //incrementing file name
		sFileName := CONCAT (STR1 := location, STR2 := filename);
		
		fbFileOpen( sNetId := sNetId, sPathName := sFileName, nMode := FOPEN_MODEWRITE OR FOPEN_MODETEXT,(* Open file in TEXT mode! *)
					ePath := PATH_GENERIC, bExecute := TRUE );
		step := 2;

	2:(* Wait until open not busy *)
		fbFileOpen( bExecute := FALSE, bError => bError, nErrID => nErrID, hFile => hFile );
		IF NOT fbFileOpen.bBusy THEN
			IF NOT fbFileOpen.bError THEN
				step := 3;
			ELSE(* Error: file not found? *)
				step := 100;
			END_IF
		END_IF

	3:(* Convert one PLC record to CSV format *)
		sCSVLine := '';
		fbWriter.eCmd := eEnumCmd_First;(* Write first field value *)
		IF nRow <= GVL.MAX_CSV_ROWS THEN
		
			FOR nColumn := 0 TO GVL.MAX_CSV_COLUMNS BY 1 DO

				sCSVField := STRING_TO_CSVFIELD( database[ nRow, nColumn ], FALSE );(* TODO: Get field value from your application *)

				(* Add new field to the record buffer *)
				fbWriter( 	pBuffer := ADR( sCSVLine ), cbBuffer := SIZEOF( sCSVLine ) - 1, putValue := sCSVField, pValue := 0, cbValue := 0,
							bCRLF := ( nColumn = GVL.MAX_CSV_COLUMNS ) );(* bCRLF == TRUE => Write CRLF after the last field value *)
				IF fbWriter.bOk THEN
					fbWriter.eCmd := eEnumCmd_Next;(* Write next field value *)
				ELSE(* Error *)
					step := 100;
					RETURN;
				END_IF

			END_FOR(* FOR nColumn := 0... *)

			(* FB_FilePuts adds allready CR (carriage return) to the written line.
			We have to replace the $R$L characters with $L character to avoid double CR. *)
			IF RIGHT( sCSVLine, 2 ) = '$R$L' THEN
				sCSVLine := REPLACE( sCSVLine, '$L', 2, LEN( sCSVLine ) - 1 );
			END_IF

			nRow := nRow + 1;(* Increment number of created records (rows) *)

			step := 4;(* Write record to the file *)

		ELSE(* All rows written => Close file *)
			step := 10;
		END_IF

	4:	(* Write single text line *)
		fbFilePuts( bExecute := FALSE );
		fbFilePuts( sNetId := sNetId, hFile := hFile, sLine := sCSVLine, bExecute := TRUE );
		step := 5;

	5:(* Wait until write not busy *)
		fbFilePuts( bExecute := FALSE, bError => bError, nErrID => nErrID );
		IF NOT fbFilePuts.bBusy THEN
			IF NOT fbFilePuts.bError THEN
				step := 3;(* Write next record *)
			ELSE(* Error *)
				step := 100;
			END_IF
		END_IF

	10:	(* Close source file *)
		fbFileClose( bExecute := FALSE );
		fbFileClose( sNetId := sNetId, hFile := hFile, bExecute := TRUE );
		step := 11;

	11:(* Wait until close not busy *)
		fbFileClose( bExecute := FALSE, bError => bError, nErrID => nErrID );
		IF ( NOT fbFileClose.bBusy ) THEN
			hFile := 0;
			step := 100;
		END_IF

	100: (* Error or ready step => cleanup *)
		IF ( hFile <> 0 ) THEN
			step := 10; (* Close the source file *)
		ELSE
			bBusy := FALSE;
			step := 0;	(* Ready *)
		END_IF

END_CASE



//logging logic
//start storing buffer when charge pb is pressed. 
//when charge done, convert data into csv.
IF (*Sequence.eState = E_State.CHARGING*) HMI_DB.ChargePB = TRUE THEN 
	//StartLogging_ONS := TRUE;
	SaveBuff := TRUE; 
	//ELSIF Sequence.eState = E_State.SAFE THEN
		//bWrite := FALSE;
		//step := 10;
		//fbFileClose( bExecute := FALSE );
		//fbFileClose( sNetId := sNetId, hFile := hFile, bExecute := TRUE );
END_IF


//logging data - either need a timer to store the database buffer or user a timer to call the function.
IF SaveBuff = TRUE THEN 
	timer_TON (IN:= TRUE, PT := (ChargeTime_DB.LongestChargeTime_PT + HMI_DB.RunOutTMR_PT + T#10S), ET => timer_ET);
	IF SamplingTMR_TON.Q = FALSE THEN
		SamplingTMR_TON (IN := TRUE, PT := SamplingTMR_PT, ET => SamplingTMR_ET);
		//csvW_RebounceTMR_TON(IN := TRUE, PT := csvW_RebounceTMR_PT );
		ELSE 
			SamplingTMR_TON (IN := FALSE, PT := SamplingTMR_PT);
	END_IF 
ELSE
		SamplingTMR_TON (IN := FALSE, PT := SamplingTMR_PT);
		timer_TON (IN:= FALSE);
END_IF

timestamp := TIME_TO_REAL (timer_ET)/1000; 
	
IF (i <= GVL.MAX_CSV_ROWS) AND SamplingTMR_TON.Q = TRUE THEN 
	database[i, 0] := REAL_TO_STRING(timestamp);
	database[i, 1] := REAL_TO_STRING(MCP_IO.MagDriver[1].ShotCurrentFeedback);
	database[i, 2] := REAL_TO_STRING(MCP_IO.MagDriver[2].ShotCurrentFeedback);
	database[i, 3] := REAL_TO_STRING(MCP_IO.MagDriver[3].ShotCurrentFeedback);	
	database[i, 4] := REAL_TO_STRING(MCP_IO.MagDriver[4].ShotCurrentFeedback);	
	database[i, 5] := REAL_TO_STRING(MCP_IO.MagDriver[5].ShotCurrentFeedback);	
	database[i, 6] := REAL_TO_STRING(MCP_IO.MagDriver[6].ShotCurrentFeedback);	
	//uncomment for testing purposes
		//Input.R1_08_00 := Input.R1_08_00 + 10 ;
		//Input.R1_08_01 := Input.R1_08_00 + 100 ;
		i := i + 1;
		SamplingTMR_TON.IN := FALSE;

ELSIF (i > GVL.MAX_CSV_ROWS) OR ((Sequence.eState = E_State.ABORT OR HMI_DB.FirePB = TRUE OR HMI_DB.DumpPB = TRUE OR HMI_DB.AbortPB = TRUE) AND i <> 0) THEN 
	SaveCSV := TRUE;
	SaveBuff := FALSE; 
	SamplingTMR_TON.IN := FALSE;
	i := 0;
	ELSE
		SamplingTMR_TON.IN := FALSE;
END_IF

